                    IF iCurrentCopyY > _RecipeBuilder.ActualCopiesY THEN
                        //Trace(Message := 'Step 90: ZAKONCZONO WSZYSTKIE KOPIE (Nesting gotowy). Skok do 1000.');
                        nStep := 1000;
                    ELSE
                        //Trace(Message := CONCAT('Step 90: Skok do nastepnego rzedu (Kopia Y): ', TO_STRING(iCurrentCopyY)));
                        iCurrentSegment := 1;
                        nStep := 10;
                    END_IF
                ELSE
                    //Trace(Message := CONCAT('Step 90: Skok do nastepnego detalu w rzedzie (Kopia X): ', TO_STRING(iCurrentCopyX)));
                    iCurrentSegment := 1;
                    nStep := 10;
                END_IF
            ELSE
                nStep := 10;
            END_IF
        END_IF

    999: // Błąd
        //Trace(Message := 'Step 999: FATAL ERROR - Aborting');
        _bBusy := FALSE; _bError := TRUE; _bDone := FALSE; nStep := 0;

    1000: // Koniec
        //Trace(Message := 'Step 1000: ZAKONCZONO CALA OPERACJE CIECIA.');
        _bBusy := FALSE; _bDone := TRUE; nStep := 0;
END_CASE
END_METHOD

END_FUNCTION_BLOCK

// ---- POUs/Executor/FB_ExecutorBase.TcPOU
FUNCTION_BLOCK FB_ExecutorBase EXTENDS FB_CyclicFB IMPLEMENTS I_MachiningExecutor, I_BB8Specification
VAR
    // Zmienne sekwencyjne 
    nStep           : INT;
    iCurrentSegment : INT;
    StepTimer       : TON;
    _bBusy          : BOOL;
    _bDone          : BOOL;
    _bError         : BOOL;
    _uErrorID       : UDINT;

    // --- ZMIENNE WSPÓLNE DLA WSZYSTKICH EXECUTORÓW
    _AxisX          : SPT_Motion_Control.I_BasicAxis;
    _AxisY          : SPT_Motion_Control.I_BasicAxis;
    _AxisZ          : SPT_Motion_Control.I_BasicAxis;
	_AxisQ			: SPT_Motion_Control.I_BasicAxis;
    _Cylinder       : I_Cylinder;                     
    _RecipeBuilder  : I_RecipeBuilder;
	_ConfigProvider : I_GantryConfigProvider;
	
	iCurrentCopyX : INT := 1;
    iCurrentCopyY : INT := 1;
END_VAR

METHOD Abort
_bBusy := FALSE;
_bDone := FALSE;
nStep := 0;
iCurrentSegment := 1;
StepTimer(IN := FALSE);
END_METHOD

PROPERTY AxisQ : I_BasicAxis
GET
AxisQ := _AxisQ;
END_GET
SET
_AxisQ := AxisQ;
END_SET
END_PROPERTY

PROPERTY AxisX : I_BasicAxis
GET
AxisX := _AxisX;
END_GET
SET
_AxisX := AxisX;
END_SET
END_PROPERTY

PROPERTY AxisY : I_BasicAxis
GET
AxisY := _AxisY;
END_GET
SET
_AxisY := AxisY;
END_SET
END_PROPERTY

PROPERTY AxisZ : I_BasicAxis
GET
AxisZ := _AxisZ;
END_GET
SET
_AxisZ := AxisZ;
END_SET
END_PROPERTY

PROPERTY Busy : BOOL
GET
Busy := _bBusy;
END_GET
END_PROPERTY

PROPERTY ConfigProvider : I_GantryConfigProvider
GET
ConfigProvider := _ConfigProvider;
END_GET
SET
_ConfigProvider := ConfigProvider;
END_SET
END_PROPERTY

METHOD PUBLIC  CyclicLogic
VAR_INPUT
END_VAR
END_METHOD

PROPERTY Cylinder : I_Cylinder
GET
Cylinder := _Cylinder;
END_GET
SET
_Cylinder := Cylinder;
END_SET
END_PROPERTY

PROPERTY Done : BOOL
GET
Done := _bDone;
END_GET
END_PROPERTY

PROPERTY Error : BOOL
GET
Error := _bError;
END_GET
END_PROPERTY


PROPERTY ErrorID : UDINT
GET
ErrorID := _uErrorID;
END_GET
END_PROPERTY

METHOD Execute : BOOL
IF _bBusy THEN RETURN; END_IF

_bBusy    := TRUE;
_bDone    := FALSE;
_bError   := FALSE;
_uErrorID := 0;
nStep     := 5; 
iCurrentCopyX := 1; 
iCurrentCopyY := 1; 
Execute   := TRUE;
END_METHOD

METHOD PROTECTED MoveToXY 
VAR_INPUT
    TargetX     : REAL; 
    TargetY     : REAL; 
    ToolOffsetX : REAL := 0.0; 
    ToolOffsetY : REAL := 0.0; 
END_VAR
VAR
    localConfig : ST_GantryXYZ_Config;
	NestingOffsetX : REAL;
    NestingOffsetY : REAL;
END_VAR
// Pobieramy bezpieczną konfigurację z Providera (zawiera GlobalOffset)
localConfig := _ConfigProvider.Config;

// Odejmujemy 1, bo pierwsza kopia (indeks 1) ma offset 0.0
NestingOffsetX := (iCurrentCopyX - 1) * _RecipeBuilder.FootprintX;
NestingOffsetY := (iCurrentCopyY - 1) * _RecipeBuilder.FootprintY;

// I dodajemy to do naszych wspaniałych komend jazdy:
_AxisX.MoveAbsolute(TargetX + ToolOffsetX + NestingOffsetX + localConfig.GlobalOffsetX, 0);
_AxisY.MoveAbsolute(TargetY + ToolOffsetY + NestingOffsetY + localConfig.GlobalOffsetY, 0);
END_METHOD

PROPERTY RecipeBuilder : I_RecipeBuilder
GET
RecipeBuilder := _RecipeBuilder;
END_GET
SET
_RecipeBuilder := RecipeBuilder;
END_SET
END_PROPERTY

END_FUNCTION_BLOCK

// ---- POUs/Executor/FB_Exec_Spindle_PTP.TcPOU
FUNCTION_BLOCK FB_Exec_Spindle_PTP EXTENDS FB_ExecutorBase

METHOD PUBLIC CyclicLogic
VAR_INST
    // Lokalne zmienne pomocnicze na czas trwania cyklu
    currentSeg          : ST_CutSegment;
    localConfig         : ST_GantryXYZ_Config;
    recipeConfig        : ST_RecipeBuilder_Config; 
    
    MaterialTopZ        : REAL;
    SafeZ               : REAL;
    TargetZ             : REAL;

    // Zmienne sekwencyjne dla logiki frezowania
    iPass               : INT;
    currentDepth        : LREAL;
    g1, g2, g3, g4, g5  : LREAL;
    v1, v2, v3, v4, v5  : LREAL;
END_VAR
StepTimer();

// Zabezpieczenie na wypadek braku wstrzykniętych referencji!
IF _RecipeBuilder = 0 OR _ConfigProvider = 0 THEN
    RETURN;
END_IF

// Pobieramy konfigurację do pamięci podręcznej 
localConfig := _ConfigProvider.Config;

IF iCurrentSegment < 1 THEN iCurrentSegment := 1; END_IF
IF iCurrentSegment > 32 THEN iCurrentSegment := 32; END_IF

// Wyciągnięcie konkretnego segmentu dla aktualnego kroku
currentSeg := _RecipeBuilder.SegmentsGroove[iCurrentSegment];

// 1. Z=0 to stół. 
// Dodajemy podkład (GlobalOffsetZ) i grubość deski (RawBoardZ).
// To daje nam absolutną pozycję górnej krawędzi płyty w układzie maszyny.
MaterialTopZ := localConfig.GlobalOffsetZ + localConfig.RawBoardZ;

// 2. Pozycja bezpieczna to wierzch płyty + prześwit (np. 10 mm).
// Na tej wysokości możemy latać na parametrze RapidSpeedZ.
SafeZ := MaterialTopZ + localConfig.SafeClearanceZ;

CASE nStep OF
    
    0: // IDLE - maszyna czeka na wywołanie Execute()

    // -------- Inicjalizacja procesu --------
    5:
        // Konfiguracja głębokości (g) i mnożników prędkości (v)
        g1 := 3.5; g2 := 3.5; g3 := 1.5; g4 := 0.0; g5 := 0.0;
        v1 := 1.0; v2 := 1.0; v3 := 1.0; v4 := 1.0; v5 := 1.0;

        IF _AxisX.Enable() AND _AxisY.Enable() AND _AxisZ.Enable() THEN
            IF _RecipeBuilder.SegmentsToGroove <= 0 THEN
                nStep := 1000;
                RETURN;
            END_IF;
           
            _AxisX.Velocity := localConfig.RapidSpeedX;
            _AxisY.Velocity := localConfig.RapidSpeedY;
            _AxisZ.Velocity := localConfig.RapidSpeedZ;

            iCurrentSegment := 1;
            iPass := 4; // Zgodnie z oryginalnym plikiem testowym
            
            IF NOT _AxisX.Busy AND NOT _AxisY.Busy AND NOT _AxisZ.Busy THEN
                nStep := 10;
            END_IF     
        END_IF

    // -------- Dojazd XY do poczatku (Start) --------
    10:
        MoveToXY(currentSeg.Start.X, currentSeg.Start.Y, 0.0, 0.0);
        nStep := 20;

    20: // Czekamy na pozycje XY
        IF _AxisX.Error OR _AxisY.Error THEN 
            nStep := 999;
        ELSIF _AxisX.InPosition AND _AxisY.InPosition THEN 
            _AxisZ.Velocity := localConfig.GroovingSpeedZ;
            nStep := 30;
        END_IF

    // -------- Wybor glebokosci dla przejsc --------
    30:
        recipeConfig := _RecipeBuilder.Config;
        
        CASE iPass OF
            1: currentDepth := recipeConfig.GrooveDepthZ - g1;
            2: currentDepth := recipeConfig.GrooveDepthZ - g2;
            3: currentDepth := recipeConfig.GrooveDepthZ - g3;
            4: currentDepth := recipeConfig.GrooveDepthZ - g4;
            5: currentDepth := recipeConfig.GrooveDepthZ - g5;
        ELSE
            currentDepth := recipeConfig.GrooveDepthZ;
        END_CASE;

        // 3. OBLICZENIE ABSOLUTNEGO CELU DLA OSI Z
        // Skoro MaterialTopZ to góra płyty, a currentDepth to to głębokość,
        // na jaką musimy się w nią zanurzyć - TargetZ = MaterialTopZ - currentDepth.
        TargetZ := MaterialTopZ - currentDepth;
        _AxisZ.MoveAbsolute(TargetZ, 0);
        nStep := 40;

    40: // Czekamy az os Z zjedzie
        IF _AxisZ.Error THEN 
            nStep := 999;
        ELSIF _AxisZ.InPosition THEN
            // Wybor predkosci posuwu roboczego w zaleznosci od przejscia
			// Wybor predkosci posuwu roboczego w zaleznosci od przejscia
            CASE iPass OF
                1: _AxisX.Velocity := localConfig.GroovingSpeedXY * v1; _AxisY.Velocity := localConfig.GroovingSpeedXY * v1;
                2: _AxisX.Velocity := localConfig.GroovingSpeedXY * v2; _AxisY.Velocity := localConfig.GroovingSpeedXY * v2;
                3: _AxisX.Velocity := localConfig.GroovingSpeedXY * v3; _AxisY.Velocity := localConfig.GroovingSpeedXY * v3;
                4: _AxisX.Velocity := localConfig.GroovingSpeedXY * v4; _AxisY.Velocity := localConfig.GroovingSpeedXY * v4;
                5: _AxisX.Velocity := localConfig.GroovingSpeedXY * v5; _AxisY.Velocity := localConfig.GroovingSpeedXY * v5;
            END_CASE;
            
            nStep := 50;
        END_IF
            
    50: // Czekanie przed ruchem
        StepTimer(IN := TRUE, PT := REAL_TO_TIME(localConfig.GroovingIdleTime * 1000.0));
        IF StepTimer.Q THEN
            StepTimer(IN := FALSE);
            nStep := 60;
        END_IF

    // -------- Frezowanie do punktu koncowego --------
    60:
        MoveToXY(currentSeg.Stop.X, currentSeg.Stop.Y, 0.0, 0.0);
        nStep := 70;

    70: // Czekamy na koniec cięcia
        IF _AxisX.Error OR _AxisY.Error OR _AxisZ.Error THEN 
            nStep := 999;
        ELSIF _AxisX.InPosition AND _AxisY.InPosition AND _AxisZ.InPosition THEN
            IF iPass = 5 THEN
                nStep := 74;
            ELSE
                _AxisZ.Velocity := localConfig.RapidSpeedZ;
                nStep := 80;
            END_IF
        END_IF

    // -------- Procedura czyszcząca na koniec 5-go przejazdu --------
    74:
        StepTimer(IN := TRUE, PT := T#500MS);
        IF StepTimer.Q THEN
            StepTimer(IN := FALSE);
            nStep := 75;
        END_IF

    75: 
        MoveToXY(currentSeg.Start.X, currentSeg.Start.Y, 0.0, 0.0);
        nStep := 76;

    76: 
        IF _AxisX.Error OR _AxisY.Error THEN 
            nStep := 999;
        ELSIF _AxisX.InPosition AND _AxisY.InPosition THEN
            _AxisZ.Velocity := localConfig.RapidSpeedZ;
            nStep := 80;
        END_IF

    // -------- Podnoszenie osi Z na pozycję bezpieczną --------
    80:
        // 4. UŻYCIE POZYCJI BEZPIECZNEJ SafeZ 
        // Wcześniej było to sztywne `0`, co stanowiło ryzyko kolizji z materiałem.
        _AxisZ.MoveAbsolute(SafeZ, 0);
        nStep := 90;

    90: 
        IF _AxisZ.Error THEN 
            nStep := 999;
        ELSIF _AxisZ.InPosition THEN
            nStep := 100;
        END_IF  

    100: // Czas stabilizacji po przejsciu
        StepTimer(IN := TRUE, PT := REAL_TO_TIME(localConfig.GroovingIdleTime * 1000.0));
        IF StepTimer.Q THEN
            StepTimer(IN := FALSE);
            
            // Powrot predkosci X/Y na rapid
            _AxisX.Velocity := localConfig.RapidSpeedX;
            _AxisY.Velocity := localConfig.RapidSpeedY;
            iCurrentSegment := iCurrentSegment + 1;
            
            // Logika zmiany przejazdu / zakonczenia
            IF iCurrentSegment > _RecipeBuilder.SegmentsToGroove THEN
                IF iPass < 5 THEN
                    iPass := iPass + 1;
                    iCurrentSegment := 1;
                    nStep := 10;
                ELSE
                    // CZYSTA PĘTLA NESTINGU (Zrobiono wszystkie 5 passów)
                    iCurrentCopyX := iCurrentCopyX + 1;
                    
                    IF iCurrentCopyX > _RecipeBuilder.ActualCopiesX THEN
                        iCurrentCopyX := 1;
                        iCurrentCopyY := iCurrentCopyY + 1;
                        
                        IF iCurrentCopyY > _RecipeBuilder.ActualCopiesY THEN
                            nStep := 1000;
                        ELSE
                            iPass := 1;
                            iCurrentSegment := 1;
                            nStep := 10;
                        END_IF
                    ELSE
                        iPass := 1;
                        iCurrentSegment := 1;
                        nStep := 10;
                    END_IF
                END_IF
            ELSE
                nStep := 10;
            END_IF
        END_IF

    999: // Błąd którejkolwiek osi
        _bBusy  := FALSE;
        _bError := TRUE; 
        _bDone  := FALSE;
        nStep   := 0;

    1000: // Zakonczenie operacji frezowania
        _bBusy := FALSE;
        _bDone := TRUE;
        nStep := 0;
END_CASE
END_METHOD

END_FUNCTION_BLOCK

// ---- POUs/Executor/FB_Exec_Drill_PTP.TcPOU
FUNCTION_BLOCK FB_Exec_Drill_PTP EXTENDS FB_ExecutorBase

METHOD PUBLIC CyclicLogic
VAR_INST
    currentHole   : ST_PointXY;
    localConfig   : ST_GantryXYZ_Config;
    recipeConfig  : ST_RecipeBuilder_Config;
    
    MaterialTopZ  : REAL;
    SafeZ         : REAL;
    TargetZ       : REAL;
END_VAR
// 1. Zabezpieczenia i cykliczny timer z klasy bazowej
StepTimer();
IF _RecipeBuilder = 0 OR _ConfigProvider = 0 OR _AxisQ = 0 THEN RETURN; END_IF

// 2. Cache'owanie danych wejściowych
localConfig := _ConfigProvider.Config;

// Zabezpieczenie zakresu tablicy
IF iCurrentSegment < 1 THEN iCurrentSegment := 1; END_IF
IF iCurrentSegment > 1000 THEN iCurrentSegment := 1000; END_IF

currentHole := _RecipeBuilder.HolesDrill[iCurrentSegment];

// 3. Oliczenie bezpiecznych poziomów w osi Z 
MaterialTopZ := localConfig.GlobalOffsetZ + localConfig.RawBoardZ;
SafeZ := MaterialTopZ + localConfig.SafeClearanceZ;

CASE nStep OF
    0: // IDLE

    5: // INIT - Aktywacja osi i przygotowanie (X, Y, Z oraz Q!)
        IF _AxisX.Enable() AND _AxisY.Enable() AND _AxisZ.Enable() AND _AxisQ.Enable() THEN
            IF _RecipeBuilder.HolesToDrill <= 0 THEN
                nStep := 1000; // Brak otworów do wiercenia
                RETURN;
            END_IF;
           
            _AxisX.Velocity := localConfig.RapidSpeedX;
            _AxisY.Velocity := localConfig.RapidSpeedY;
            _AxisZ.Velocity := localConfig.RapidSpeedZ;
            _AxisQ.Velocity := localConfig.RapidSpeedQ; // Ustawienie prędkosci noża

            iCurrentSegment := 1;
            nStep := 6;
      END_IF
	  
	6:
		IF NOT _AxisX.Busy AND NOT _AxisY.Busy AND NOT _AxisZ.Busy AND NOT _AxisQ.Busy THEN
			nStep := 10;
		END_IF   

    // -------- Dojazd XY nad punkt otworu --------
    10:
        MoveToXY(currentHole.X, currentHole.Y, 0.0, 0.0);
        nStep := 20;

    20: // Czekamy na pozycje XY
        IF _AxisX.Error OR _AxisY.Error THEN 
            nStep := 999;
        ELSIF _AxisX.InPosition AND _AxisY.InPosition THEN 
            // Ustawiamy prędkość roboczą dla zagłębiania noża
            _AxisZ.Velocity := localConfig.GroovingSpeedZ;
            nStep := 30;
        END_IF

    // -------- Zjazd Z (Zanurzenie noża w gąbce) --------
    30:
        recipeConfig := _RecipeBuilder.Config;
        TargetZ := MaterialTopZ - 2.0;
        _AxisZ.MoveAbsolute(TargetZ, 0);
        nStep := 40;

    40: // Czekamy aż nóż wejdzie w materiał
        IF _AxisZ.Error THEN 
            nStep := 999;
        ELSIF _AxisZ.InPosition THEN
            // Zjechaliśmy! Teraz kręcimy nożem tangencjalnym do 720 stopni
            _AxisQ.MoveAbsolute(720.0, 0);
            nStep := 42;
        END_IF
        
    // -------- Obrót Q: Piruet otworowy --------
    42: // Czekamy aż nóż osiągnie +720 stopni
        IF _AxisQ.Error THEN
            nStep := 999;
        ELSIF _AxisQ.InPosition THEN
            // Wracamy nożem do 0 stopni, żeby nie zrywać przewodów/pasków
            _AxisQ.MoveAbsolute(0.0, 0);
            nStep := 44;
        END_IF
        
    44: // Czekamy aż nóż wróci do 0
        IF _AxisQ.Error THEN
            nStep := 999;
        ELSIF _AxisQ.InPosition THEN
            nStep := 50;
        END_IF
            
    50: // Czekanie na dnie otworu (Opcjonalne uspokojenie materiału po obrocie)
        StepTimer(IN := TRUE, PT := REAL_TO_TIME(localConfig.GroovingIdleTime * 1000.0));
        IF StepTimer.Q THEN
            StepTimer(IN := FALSE);
            nStep := 60;
        END_IF

    // -------- Szybki wyjazd z materiału --------
    60:
        _AxisZ.Velocity := localConfig.RapidSpeedZ;
        _AxisZ.MoveAbsolute(SafeZ, 0);
        nStep := 70;

    70: // Czekamy na wyjazd osi Z
        IF _AxisZ.Error THEN 
            nStep := 999;
        ELSIF _AxisZ.InPosition THEN
            // Krok zakończony - idziemy do następnego otworu
            iCurrentSegment := iCurrentSegment + 1;
            
            IF iCurrentSegment > _RecipeBuilder.HolesToDrill THEN
                // CZYSTA PĘTLA NESTINGU
                iCurrentCopyX := iCurrentCopyX + 1;
                
                IF iCurrentCopyX > _RecipeBuilder.ActualCopiesX THEN
                    iCurrentCopyX := 1;
                    iCurrentCopyY := iCurrentCopyY + 1;
                    
                    IF iCurrentCopyY > _RecipeBuilder.ActualCopiesY THEN
                        // Wiercenie wszystkich kopii zakończone
                        nStep := 1000;
                    ELSE
                        iCurrentSegment := 1;
                        nStep := 10;
                    END_IF
                ELSE
                    iCurrentSegment := 1;
                    nStep := 10;
                END_IF
            ELSE
                nStep := 10;
            END_IF
        END_IF

    // -------- Awaria --------
    999: 
        _bBusy  := FALSE;
        _bError := TRUE; 
        _bDone  := FALSE;
        nStep   := 0;
        
    // -------- Sukces --------
    1000: 
        _bBusy := FALSE;
        _bDone := TRUE;
        nStep := 0;
END_CASE
END_METHOD

END_FUNCTION_BLOCK

// ---- POUs/Executor/FB_Exec_Tangential_FeedTable.TcPOU
FUNCTION_BLOCK FB_Exec_Tangential_FeedTable EXTENDS FB_ExecutorBase IMPLEMENTS I_GeometryWriter
VAR
    _NciChannel : I_NciChannel_FeedTable;
    _FeedTable  : ST_NciFeedGroupTable; 
    
    // NCI Builder z Tc2_PlcInterpolation
    fbFeedPrep  : FB_NciFeedTablePreparation;
	
	// Lokalne offsety aktualizowane co kopię nestingu
	_CurrentOffsetX : LREAL;
	_CurrentOffsetY : LREAL;
END_VAR

METHOD Abort
IF _NciChannel <> 0 THEN
    _NciChannel.Stop();
    _NciChannel.ResetChannel();
    _NciChannel.Ungroup();
END_IF
_bBusy := FALSE; _bDone := FALSE; _bError := FALSE; _uErrorID := 0; nStep := 0;
END_METHOD

METHOD AddArc : BOOL
VAR_INPUT
    TargetX    : LREAL;
    TargetY    : LREAL;
    CenterX    : LREAL;
    CenterY    : LREAL;
    Velo       : LREAL;
    Clockwise  : BOOL; 
END_VAR
VAR
    stArc : ST_NciGeoCirclePlane;
END_VAR
stArc.fEndPosX := TargetX + _CurrentOffsetX;
stArc.fEndPosY := TargetY + _CurrentOffsetY;
stArc.fCenterX := CenterX + _CurrentOffsetX;
stArc.fCenterY := CenterY + _CurrentOffsetY;
stArc.fVelo := Velo;
stArc.bClockwise := Clockwise;
stArc.nPlane := E_NciGeoPlane.E_NciGeoPlaneXY;

fbFeedPrep(
    nEntryType := E_NciEntryType.E_NciEntryTypeGeoCirclePlane,
    pEntry := ADR(stArc),
    bResetTable := FALSE,
    bResetAll := FALSE,
    stFeedGroupTable := _FeedTable
);
AddArc := NOT fbFeedPrep.bError;
END_METHOD

METHOD AddLine : BOOL
VAR_INPUT
    TargetX : LREAL;
    TargetY : LREAL;
    Velo    : LREAL;
END_VAR
VAR
    stLine : ST_NciGeoLine;
END_VAR
stLine.fEndPosX := TargetX + _CurrentOffsetX;
stLine.fEndPosY := TargetY + _CurrentOffsetY;
stLine.fVelo := Velo;

fbFeedPrep(
    nEntryType := E_NciEntryType.E_NciEntryTypeGeoLine,
    pEntry := ADR(stLine),
    bResetTable := FALSE,
    bResetAll := FALSE,
    stFeedGroupTable := _FeedTable
);
AddLine := NOT fbFeedPrep.bError;
END_METHOD

METHOD AddStartPoint : BOOL
VAR_INPUT
    TargetX : LREAL;
    TargetY : LREAL;
END_VAR
VAR
    stStart : ST_NciGeoStart;
END_VAR
stStart.fPosX := TargetX + _CurrentOffsetX;
stStart.fPosY := TargetY + _CurrentOffsetY;

fbFeedPrep(
    nEntryType := E_NciEntryType.E_NciEntryTypeGeoStart,
    pEntry := ADR(stStart),
    bResetTable := FALSE,
    bResetAll := FALSE,
    stFeedGroupTable := _FeedTable
);
AddStartPoint := NOT fbFeedPrep.bError;
END_METHOD

METHOD Clear : BOOL
VAR_INPUT
END_VAR
fbFeedPrep(
    nEntryType := E_NciEntryType.E_NciEntryTypeNone,
    pEntry := 0,
    bResetTable := TRUE,
    bResetAll := TRUE, // Czyści też modale i błędy (wg str. 315)
    stFeedGroupTable := _FeedTable
);
Clear := NOT fbFeedPrep.bError;
END_METHOD

METHOD PUBLIC CyclicLogic
VAR_INST
    localConfig   : ST_GantryXYZ_Config;
    recipeConfig  : ST_RecipeBuilder_Config;
    MaterialTopZ  : REAL;
    SafeZ         : REAL;
    TargetZ       : REAL;
    iCurrentShape : INT := 1;
END_VAR
SUPER^.CyclicLogic();

IF nStep > 0 THEN
    IF _RecipeBuilder = 0 OR _ConfigProvider = 0 OR _NciChannel = 0 THEN
        nStep := 999;
    END_IF
END_IF

CASE nStep OF
    0: 
		;
    5: 
        IF _AxisX.Enable() AND _AxisY.Enable() AND _AxisZ.Enable() AND _AxisQ.Enable() THEN
            IF _AxisX.Enabled AND _AxisY.Enabled AND _AxisZ.Enabled AND _AxisQ.Enabled 
               AND NOT _AxisX.Busy AND NOT _AxisY.Busy AND NOT _AxisQ.Busy THEN
                
                _bBusy := TRUE;
                localConfig := _ConfigProvider.Config;
                recipeConfig := _RecipeBuilder.Config;

                IF NOT recipeConfig.IsValid THEN
                    nStep := 1000;
                    RETURN;
                END_IF

                iCurrentCopyX := 1;
                iCurrentCopyY := 1;
                iCurrentShape := 1;

                _AxisX.Velocity := localConfig.RapidSpeedX;
                _AxisY.Velocity := localConfig.RapidSpeedY;
                _AxisZ.Velocity := localConfig.RapidSpeedZ;
                _AxisQ.Velocity := localConfig.RapidSpeedQ;

                nStep := 8;
            END_IF
        END_IF

    8: 
        localConfig := _ConfigProvider.Config;
		_CurrentOffsetX := (iCurrentCopyX - 1) * _RecipeBuilder.FootprintX + localConfig.GlobalOffsetX;
		_CurrentOffsetY := (iCurrentCopyY - 1) * _RecipeBuilder.FootprintY + localConfig.GlobalOffsetY;
		
        _RecipeBuilder.CurrentShapeIndex := iCurrentShape;
		_RecipeBuilder.Build();
		nStep := 85;

	85:
		IF _RecipeBuilder.Done THEN
			recipeConfig := _RecipeBuilder.Config;
			MoveToXY(_RecipeBuilder.ShapeStart[iCurrentShape].X, _RecipeBuilder.ShapeStart[iCurrentShape].Y, 0.0, 0.0);
			_AxisQ.MoveAbsolute(0.0, 0);
			nStep := 9;
		ELSIF _RecipeBuilder.Error THEN
			nStep := 999;
		END_IF

    9: 
        IF _AxisX.Error OR _AxisY.Error OR _AxisZ.Error OR _AxisQ.Error THEN
            nStep := 999;
        ELSIF _AxisX.InPosition AND _AxisY.InPosition AND NOT _AxisQ.Busy THEN
            localConfig := _ConfigProvider.Config;
            MaterialTopZ := localConfig.GlobalOffsetZ + localConfig.RawBoardZ;
            SafeZ := MaterialTopZ + localConfig.SafeClearanceZ;

            IF _AxisZ.MoveAbsolute(SafeZ, 0) THEN
                nStep := 10;
            END_IF
        END_IF

    10: 
        IF _AxisZ.Error THEN
            nStep := 999;
        ELSIF _AxisZ.InPosition THEN
            nStep := 20;
        END_IF

    20: 
        _NciChannel.BuildGroup();
        nStep := 30;

    30: 
        IF _NciChannel.ChannelError THEN
            nStep := 999;
        ELSIF _NciChannel.IsGrouped THEN
            TargetZ := MaterialTopZ - recipeConfig.GrooveDepthZ;
            _AxisZ.Velocity := localConfig.GroovingSpeedZ;
			IF  _AxisZ.MoveAbsolute(TargetZ, 0) THEN
				nStep := 35;
			END_IF
        END_IF

    35: 
        IF _AxisZ.Error THEN
            nStep := 999;
        ELSIF _AxisZ.InPosition THEN
            _NciChannel.StartFeedTable(stTable := THIS^._FeedTable); 
            nStep := 40;
        END_IF

    40: 
        IF _NciChannel.ChannelError THEN
            nStep := 999;
        ELSIF _NciChannel.IsFeedingDone THEN
            nStep := 50;
        END_IF

    50: 
        IF _NciChannel.ChannelError THEN
            nStep := 999;
        ELSIF _NciChannel.IsChannelDone THEN
            _AxisZ.Velocity := localConfig.RapidSpeedZ;
            _AxisZ.MoveAbsolute(SafeZ, 0);
            nStep := 55;
        END_IF

    55:
        IF _AxisZ.Error THEN
            nStep := 999;
        ELSIF _AxisZ.InPosition THEN
            _NciChannel.ResetChannel();
            nStep := 80;
        END_IF

    80: 
        _NciChannel.Ungroup();
        nStep := 90;

    90: 
        IF NOT _NciChannel.IsGrouped THEN
            iCurrentShape := iCurrentShape + 1;
            IF iCurrentShape > _RecipeBuilder.ShapesCount THEN
                iCurrentShape := 1;
                nStep := 110;
            ELSE
                nStep := 8;
            END_IF
        END_IF

    110:
        iCurrentCopyX := iCurrentCopyX + 1;
        IF iCurrentCopyX > _RecipeBuilder.ActualCopiesX THEN
            iCurrentCopyX := 1;
            iCurrentCopyY := iCurrentCopyY + 1;
            IF iCurrentCopyY > _RecipeBuilder.ActualCopiesY THEN
                nStep := 1000;
            ELSE
                nStep := 8;
            END_IF
        ELSE
            nStep := 8;
        END_IF

    999: 
        _bBusy := FALSE;
        _bError := TRUE;
        _bDone := FALSE;
        _uErrorID := _NciChannel.ChannelErrorId;
        _NciChannel.Ungroup();
        nStep := 0;

    1000: 
        _bBusy := FALSE;
        _bDone := TRUE;
        nStep := 0;
END_CASE
END_METHOD

METHOD EnableTangentialFollowing : BOOL
VAR
    stTf : ST_NciTangentialFollowingDesc;
END_VAR
stTf.bTangOn := TRUE;
stTf.nTangAxis := E_NciAxesInGroup.Q1Axis;
stTf.nPathAxis1 := E_NciAxesInGroup.XAxis;
stTf.nPathAxis2 := E_NciAxesInGroup.YAxis;
stTf.fOffset := -90.0;
stTf.fCriticalAngle1 := 90.0; 
stTf.nTfBehavior := E_TangentialFollowingBehavior.E_TfIngoreAll; // Uwaga na literówkę Beckhoffa!

fbFeedPrep(
    nEntryType := E_NciEntryType.E_NciEntryTypeTfDesc,
    pEntry := ADR(stTf),
    bResetTable := FALSE,
    bResetAll := FALSE,
    stFeedGroupTable := _FeedTable
);
EnableTangentialFollowing := NOT fbFeedPrep.bError;
END_METHOD

METHOD EndTable : BOOL
VAR
    stEnd : ST_NciEndOfTables;
END_VAR

fbFeedPrep(
    nEntryType := E_NciEntryType.E_NciEntryTypeEndOfTables,
    pEntry := ADR(stEnd),
    bResetTable := FALSE,
    bResetAll := FALSE,
    stFeedGroupTable := _FeedTable
);
EndTable := NOT fbFeedPrep.bError;
END_METHOD

PROPERTY NciChannel : I_NciChannel_FeedTable
GET
NciChannel := _NciChannel;
END_GET
SET
_NciChannel := NciChannel;
END_SET
END_PROPERTY

END_FUNCTION_BLOCK

// ---- POUs/Executor/FB_Exec_Spindle_GCodeXYZ.TcPOU
FUNCTION_BLOCK FB_Exec_Spindle_GCodeXYZ EXTENDS FB_ExecutorBase
VAR
    _NciChannel : I_NciChannel_GCode;
END_VAR

METHOD Abort
// 1. Zatrzymujemy program NCI (jeśli jedzie)
_NciChannel.Stop();

// 2. Wymuszamy reset błędów na kanale interpolacyjnym
_NciChannel.ResetChannel();

// 3. Dopiero teraz bezpiecznie nakazujemy kanałowi rozpięcie grupy
_NciChannel.Ungroup();

// 4. Zerujemy resztę lokalnych zmiennych Executora
_bBusy := FALSE;
_bDone := FALSE;
_bError := FALSE;
_uErrorID := 0;
nStep := 0;
iCurrentSegment := 1;
StepTimer(IN := FALSE);
END_METHOD

METHOD PUBLIC CyclicLogic
VAR_INST

    refX : Tc2_MC2.AXIS_REF;
    refY : Tc2_MC2.AXIS_REF;
    refZ : Tc2_MC2.AXIS_REF;
    
	MaterialTopZ : REAL;
    SafeZ        : REAL;

    recipeConfig  : ST_RecipeBuilder_Config;
    machineConfig : ST_GantryXYZ_Config;
END_VAR
// --- LOGIKA ---
StepTimer();

// Zabezpieczenie przed brakiem wstrzykniętych referencji
IF nStep > 0 THEN
	IF _RecipeBuilder = 0 OR _ConfigProvider = 0 OR _NciChannel = 0 OR _AxisX = 0 OR _AxisY = 0 OR _AxisZ = 0 OR _AxisQ = 0 THEN
		IF nStep > 0 THEN
			ADSLOGSTR(ADSLOG_MSGTYPE_ERROR, 'ExecutorNCI: BRAK KRYTYCZNYCH REFERENCJI (Builder/Provider/NCI/Osie)!', '');
			nStep := 999;
		END_IF
		RETURN; 
	END_IF
END_IF

CASE nStep OF
    0: // IDLE

	5: // INIT - Załączanie osi i start
		IF _AxisX.Enable() AND _AxisY.Enable() AND _AxisZ.Enable() AND _AxisQ.Enable() THEN 
			IF _AxisX.Error OR _AxisY.Error OR _AxisZ.Error OR _AxisQ.Error THEN 
				nStep := 999;
			ELSIF _AxisX.Enabled AND _AxisY.Enabled AND _AxisZ.Enabled AND _AxisQ.Enabled THEN 
				_bBusy := TRUE;
								 
				// Odczyt właściwości (Properties) do lokalnych zmiennych pomocniczych!
				machineConfig := _ConfigProvider.Config;
				recipeConfig  := _RecipeBuilder.Config;
								 
				// Bezpieczne użycie zmiennych lokalnych
				_AxisX.Velocity := machineConfig.RapidSpeedX;
				_AxisY.Velocity := machineConfig.RapidSpeedY;
				_AxisZ.Velocity := machineConfig.RapidSpeedZ;
				_AxisQ.Velocity := machineConfig.RapidSpeedQ; // <-- DODANO Q
											 
				nStep := 8;
			END_IF
		END_IF

	8: // 1. Dojazd PTP do punktu startowego NCI
       
        nStep := 9;

	9: 
		IF _AxisX.Error OR _AxisY.Error OR _AxisZ.Error OR _AxisQ.Error THEN 
			nStep := 999;
		ELSIF _AxisX.InPosition AND _AxisY.InPosition THEN
			
			machineConfig := _ConfigProvider.Config;
			
			_AxisQ.MoveAbsolute(0,0);

			nStep := 10;
		END_IF
        
    10: // Czekamy aż podniesie się Z
        IF _AxisQ.Error THEN
            nStep := 999;
        ELSIF _AxisQ.InPosition THEN
            nStep := 20;
        END_IF

	20: // 2. Zbudowanie grupy NCI
		_NciChannel.BuildGroup();
		nStep := 30;

    30: // Czekamy na spięcie osi
        IF _NciChannel.ChannelError THEN 
            nStep := 999;
        ELSIF _NciChannel.IsGrouped THEN 
            nStep := 40; 
        END_IF

    40: // 3. Załadowanie pliku G-Code
        recipeConfig := _RecipeBuilder.Config;
        _NciChannel.LoadProgram(recipeConfig.GCodePath);
        nStep := 50;

    50: // Czekamy na załadowanie do bufora
        IF _NciChannel.ChannelError THEN 
            nStep := 999;
        ELSIF _NciChannel.IsProgramLoaded THEN 
            nStep := 60;
        END_IF

    60: // 4. START programu CNC!
        _NciChannel.Start();
        StepTimer(IN:=FALSE);
        nStep := 70;
	
	70: // 4. Czekamy na koniec programu (M30)
        IF _NciChannel.ChannelError THEN 
            nStep := 999;
        ELSIF _NciChannel.IsReady THEN 
            ADSLOGSTR(ADSLOG_MSGTYPE_HINT, 'Executor: Program NCI zakonczony (M30). Rozpinam grupe...', '');
            nStep := 80;
        END_IF

    80: // 5. Rozwiązanie grupy, uwalniamy osie z powrotem do trybu PTP
        _NciChannel.Ungroup();
        nStep := 90;

	90: // 6. Reset kanału i zakończenie pracy
        IF NOT _NciChannel.IsGrouped THEN
            ADSLOGSTR(ADSLOG_MSGTYPE_HINT, 'Executor: Osie uwolnione do trybu PTP. Resetuje kanal.', '');
            _NciChannel.ResetChannel(); 
            
            nStep := 1000; 
        END_IF
        
    999: // ERROR HANDLING
        _bBusy := FALSE;
        _bError := TRUE;
        _bDone := FALSE;
        _uErrorID := _NciChannel.ChannelErrorId;
        ADSLOGDINT(ADSLOG_MSGTYPE_ERROR, 'Executor: BLAD KRYTYCZNY NCI! Kod bledu: %d', UDINT_TO_DINT(_uErrorID));
        _NciChannel.Ungroup();
        nStep := 0;

    1000: // ZAKOŃCZONO SUKCESEM
        ADSLOGSTR(ADSLOG_MSGTYPE_HINT, 'ExecutorNCI: Program wykonany pomyslnie.', '');
        _bBusy := FALSE;
        _bDone := TRUE;
        nStep := 0;

END_CASE
END_METHOD

PROPERTY NciChannel : I_NciChannel_GCode
GET
NciChannel := _NciChannel;
END_GET
SET
_NciChannel := NciChannel;
END_SET
END_PROPERTY

END_FUNCTION_BLOCK

// ---- POUs/Components/FB_NciChannel.TcPOU
FUNCTION_BLOCK FB_NciChannel EXTENDS FB_ComponentBase IMPLEMENTS I_NciChannel_GCode

VAR_INPUT
    stAxisIds : ST_NciAxisIds;
	nGroupId  : UDINT := 4;
END_VAR

VAR
    // Zmienne zlinkowane bezpośrednio z hardwarem kanału NCI
    stNciToPlc AT %I* : NCTOPLC_NCICHANNEL_REF; 
    stPlcToNci AT %Q* : PLCTONC_NCICHANNEL_REF;

    // Bloki systemowe Beckhoffa do obsługi grupy
	fbBuildExtGroup : CfgBuildExt3DGroup;
    fbUngroup       : CfgReconfigGroup;
    
    // Bloki systemowe do obsługi programu i ruchu (nowe wersje Ex)
    fbLoadProg      : ItpLoadProgEx;
    fbStartStop     : ItpStartStopEx;
    fbReset         : ItpResetEx2;
    
    _IsGrouped      : BOOL;
    _IsProgLoaded   : BOOL;
    _IsReady		:BOOL;
	


END_VAR

METHOD BuildGroup
_IsGrouped := FALSE;
_Error := FALSE; 
_ErrorId := 0;

fbBuildExtGroup(
    bExecute := TRUE,
    nGroupId := nGroupId,
    nXAxisId := stAxisIds.nX,
    nYAxisId := stAxisIds.nY,
    nZAxisId := stAxisIds.nZ,
    nQ1AxisId := stAxisIds.nQ1
);
END_METHOD

PROPERTY ChannelError : BOOL
GET
ChannelError := _Error OR (stNciToPlc.ErrorCode <> 0);
END_GET
END_PROPERTY

PROPERTY ChannelErrorId : UDINT
GET
IF stNciToPlc.ErrorCode <> 0 THEN
    ChannelErrorId := stNciToPlc.ErrorCode;
ELSE
    ChannelErrorId := _ErrorId;
END_IF
END_GET
END_PROPERTY

// This method serves as the entry point for all underlying FB logic
METHOD PUBLIC CyclicLogic

// This method should be called cyclically by descendant function blocks by invoking SUPER^.CyclicLogic().  Alternatively, the contents of this method could be reimplemented entirely in which case a call to this method would not be necessary.
// Wywołanie bazowe
SUPER^.CyclicLogic();

// Odblokowanie posuwu kanału NCI (1000000 = 100%)
stPlcToNci.ChnAxesOvr := 1000000;

// --- ODŚWIEŻANIE BLOKÓW SYSTEMOWYCH ---
fbBuildExtGroup(tTimeOut := T#2S);
fbUngroup(tTimeOut := T#2S);


fbLoadProg(
    sNciToPlc := stNciToPlc, 
    tTimeOut := T#2S
);

fbStartStop(
    sNciToPlc := stNciToPlc, 
    tTimeOut := T#2S
);

fbReset(
    sNciToPlc := stNciToPlc, 
    tTimeOut := T#2S
);

// --- AKTUALIZACJA STATUSÓW ---
// Obsługa stanów dla tworzenia grupy
IF fbStartStop.bErr THEN
    _Error := TRUE;
    _ErrorId := fbStartStop.nErrId;
    fbStartStop(bStart := FALSE, bStop := FALSE, sNciToPlc := stNciToPlc);
ELSIF fbStartStop.bBusy THEN
    // Skoro kanał NCI przyjął komendę i jest zajęty, opuszczamy Start, 
    // aby przygotować blok na kolejne uruchomienie w przyszłości
    fbStartStop(bStart := FALSE, sNciToPlc := stNciToPlc);
ELSIF NOT fbStartStop.bBusy AND fbStartStop.bStop THEN
    // Jak się poprawnie zatrzymał, opuszczamy flagę Stop
    fbStartStop(bStop := FALSE, sNciToPlc := stNciToPlc);
END_IF

// Obsługa stanów dla rozpinania grupy
IF fbUngroup.bErr THEN
    _Error := TRUE;
    _ErrorId := fbUngroup.nErrId;
    fbUngroup(bExecute := FALSE);
    _IsGrouped := FALSE; // W razie błędu awaryjnie zdejmujemy flagę, żeby maszyna nie utknęła na zawsze
ELSIF fbUngroup.bBusy = FALSE AND fbUngroup.bExecute THEN
    _IsGrouped := FALSE; // Pomyślnie rozpięto!
    fbUngroup(bExecute := FALSE);
END_IF


IF fbBuildExtGroup.bErr THEN
    _Error := TRUE;
    _ErrorId := fbBuildExtGroup.nErrId;
ELSIF fbBuildExtGroup.bBusy = FALSE AND fbBuildExtGroup.bExecute THEN
    _IsGrouped := TRUE;
    fbBuildExtGroup(bExecute := FALSE);
END_IF

// Podobnie dla ładowania programu
IF fbLoadProg.bErr THEN
    _Error := TRUE;
    _ErrorId := fbLoadProg.nErrId;
ELSIF fbLoadProg.bBusy = FALSE AND fbLoadProg.bExecute THEN
    _IsProgLoaded := TRUE;
	fbLoadProg(bExecute := FALSE, sNciToPlc := stNciToPlc);
END_IF

// --- OBSŁUGA ZEROWANIA fbReset ---
IF fbReset.bErr THEN
    _Error := TRUE;
    _ErrorId := fbReset.nErrId;
    fbReset(bExecute := FALSE, sNciToPlc := stNciToPlc);
ELSIF fbReset.bBusy = FALSE AND fbReset.bExecute THEN
    fbReset(bExecute := FALSE, sNciToPlc := stNciToPlc);
END_IF
END_METHOD

PROPERTY IsGrouped : BOOL
GET
IsGrouped := _IsGrouped;
END_GET
END_PROPERTY

PROPERTY IsMoving : BOOL
GET
IsMoving := (stNciToPlc.ItpState = 5);
END_GET
END_PROPERTY

PROPERTY IsProgramLoaded : BOOL
GET
IsProgramLoaded := _IsProgLoaded;
END_GET
END_PROPERTY

PROPERTY IsReady : BOOL
GET
IsReady := (stNciToPlc.ItpState = 2);
END_GET
END_PROPERTY

METHOD LoadProgram
VAR_INPUT
	sProgramPath : STRING(255);
END_VAR
_IsProgLoaded := FALSE;
fbLoadProg(
    bExecute := TRUE,
    sPrg := sProgramPath,
    nLength := INT_TO_UDINT(LEN(sProgramPath)),
    sNciToPlc := stNciToPlc 
);
END_METHOD

METHOD ResetChannel
VAR_INPUT
END_VAR
// Najpierw bezwarunkowo ubijamy flagi ruchu
fbStartStop(bStart := FALSE, bStop := FALSE, sNciToPlc := stNciToPlc);

// Następnie resetujemy sam kanał NCI
fbReset(
    bExecute := TRUE,
    sNciToPlc := stNciToPlc
);

_Error := FALSE;
_ErrorId := 0;
END_METHOD

METHOD Start
VAR_INPUT
END_VAR
fbStartStop(
    bStart := TRUE, 
    bStop := FALSE,
    sNciToPlc := stNciToPlc 
);
END_METHOD

METHOD Stop
VAR_INPUT
END_VAR
fbStartStop(
    bStart := FALSE, 
    bStop := TRUE,
    sNciToPlc := stNciToPlc
);
END_METHOD

METHOD Ungroup
VAR_INPUT
END_VAR
fbUngroup(
    bExecute := TRUE, 
    nGroupId := nGroupId
);
END_METHOD

END_FUNCTION_BLOCK

// ---- POUs/Components/FB_NciChannelTangential.TcPOU
FUNCTION_BLOCK FB_NciChannelTangential EXTENDS FB_ComponentBase IMPLEMENTS I_NciChannel_FeedTable

VAR_INPUT
    stAxisIds : ST_NciAxisIds;
	nGroupId  : UDINT := 5;
END_VAR

VAR
    stNciToPlc AT %I* : NCTOPLC_NCICHANNEL_REF;
    stPlcToNci AT %Q* : PLCTONC_NCICHANNEL_REF;
	
    // ZMIANA: Blok Ext3DGroup pozwala dodać osie Q1..Q5
    fbBuildExtGroup : CfgBuildExt3DGroup;
    fbUngroup       : CfgReconfigGroup;
    
    // Obsługa Resetu / Start / Stop
    fbStartStop     : ItpStartStopEx;
    fbReset         : ItpResetEx2;

    // --- NOWOŚĆ: Blok do przesyłania tabel z RAMu ---
    fbFeedTable     : FB_NciFeedTable;
    refFeedTable    : REFERENCE TO ST_NciFeedGroupTable; // Przechowuje wskaźnik do tabeli z Executora
    _bExecuteFeed   : BOOL;
    _IsFeedingDone  : BOOL;
    _IsChannelDone  : BOOL;

    _IsGrouped      : BOOL;
    _IsReady		: BOOL;
	
	_bResetFeed : BOOL;
END_VAR

METHOD BuildGroup
_IsGrouped := FALSE;
_Error := FALSE; 
_ErrorId := 0;

fbBuildExtGroup(
    bExecute := TRUE,
    nGroupId := nGroupId,
    nXAxisId := stAxisIds.nX,
    nYAxisId := stAxisIds.nY,
    nZAxisId := stAxisIds.nZ,
    nQ1AxisId := stAxisIds.nQ1 
);
END_METHOD

PROPERTY ChannelError : BOOL
GET
ChannelError := _Error OR (stNciToPlc.ErrorCode <> 0);
END_GET
END_PROPERTY

PROPERTY ChannelErrorId : UDINT
GET
IF stNciToPlc.ErrorCode <> 0 THEN
    ChannelErrorId := stNciToPlc.ErrorCode;
ELSE
    ChannelErrorId := _ErrorId;
END_IF
END_GET
END_PROPERTY

METHOD PUBLIC CyclicLogic
SUPER^.CyclicLogic();


stPlcToNci.ChnAxesOvr := 1000000;


fbBuildExtGroup(tTimeOut := T#2S);
fbUngroup(tTimeOut := T#2S);
fbStartStop(sNciToPlc := stNciToPlc, tTimeOut := T#2S);
fbReset(sNciToPlc := stNciToPlc, tTimeOut := T#2S);


IF __ISVALIDREF(refFeedTable) THEN
    fbFeedTable(
        bExecute := _bExecuteFeed,
        bReset := _bResetFeed,
        stFeedGroupTable := refFeedTable,
        stNciToPlc := stNciToPlc,
        bFeedingDone => _IsFeedingDone,
        bChannelDone => _IsChannelDone
    );
    
 
    IF _bResetFeed THEN
        _bResetFeed := FALSE;
    END_IF


    IF _IsChannelDone OR fbFeedTable.bError THEN
        IF _bExecuteFeed AND _IsChannelDone THEN
            ADSLOGSTR(ADSLOG_MSGTYPE_HINT, 'NciChannelTan: Ruch interpolowany zakonczony (Channel Done).', '');
        END_IF
        _bExecuteFeed := FALSE;
    END_IF
    
    IF fbFeedTable.bError THEN
        IF NOT _Error THEN
            ADSLOGDINT(ADSLOG_MSGTYPE_ERROR, 'NciChannelTan: BLAD FeedTable! Kod: %d', UDINT_TO_DINT(fbFeedTable.nErrorId));
        END_IF
        _Error := TRUE;
        _ErrorId := fbFeedTable.nErrorId;
    END_IF
END_IF


IF fbStartStop.bErr THEN
    IF NOT _Error THEN
        ADSLOGDINT(ADSLOG_MSGTYPE_ERROR, 'NciChannelTan: BLAD StartStop! Kod: %d', UDINT_TO_DINT(fbStartStop.nErrId));
    END_IF
    _Error := TRUE;
    _ErrorId := fbStartStop.nErrId;
    fbStartStop(bStart := FALSE, bStop := FALSE, sNciToPlc := stNciToPlc);
ELSIF fbStartStop.bBusy THEN
    fbStartStop(bStart := FALSE, sNciToPlc := stNciToPlc);
ELSIF NOT fbStartStop.bBusy AND fbStartStop.bStop THEN
    fbStartStop(bStop := FALSE, sNciToPlc := stNciToPlc);
END_IF


IF fbUngroup.bErr THEN
    IF fbUngroup.bExecute THEN
        ADSLOGDINT(ADSLOG_MSGTYPE_ERROR, 'NciChannelTan: BLAD rozpinania grupy! Kod: %d', UDINT_TO_DINT(fbUngroup.nErrId));
    END_IF
    _Error := TRUE;
    _ErrorId := fbUngroup.nErrId;
    fbUngroup(bExecute := FALSE);
    _IsGrouped := FALSE;
ELSIF fbUngroup.bBusy = FALSE AND fbUngroup.bExecute THEN
    ADSLOGSTR(ADSLOG_MSGTYPE_HINT, 'NciChannelTan: Grupa rozpieta pomyslnie.', '');
    _IsGrouped := FALSE;
    fbUngroup(bExecute := FALSE);
END_IF

IF fbBuildExtGroup.bErr THEN
    IF fbBuildExtGroup.bExecute THEN
        ADSLOGDINT(ADSLOG_MSGTYPE_ERROR, 'NciChannelTan: BLAD budowania grupy rozszerzonej! Kod: %d', UDINT_TO_DINT(fbBuildExtGroup.nErrId));
    END_IF
    _Error := TRUE;
    _ErrorId := fbBuildExtGroup.nErrId;
    fbBuildExtGroup(bExecute := FALSE); 
ELSIF fbBuildExtGroup.bBusy = FALSE AND fbBuildExtGroup.bExecute THEN
    ADSLOGSTR(ADSLOG_MSGTYPE_HINT, 'NciChannelTan: Grupa rozszerzona (X,Y,Z,Q) zbudowana pomyslnie.', '');
    _IsGrouped := TRUE;
    fbBuildExtGroup(bExecute := FALSE);
END_IF

IF fbReset.bErr THEN
    _Error := TRUE;
    _ErrorId := fbReset.nErrId;
    fbReset(bExecute := FALSE, sNciToPlc := stNciToPlc);
ELSIF fbReset.bBusy = FALSE AND fbReset.bExecute THEN
    fbReset(bExecute := FALSE, sNciToPlc := stNciToPlc);
END_IF
END_METHOD

PROPERTY IsChannelDone : BOOL
GET
IsChannelDone := _IsChannelDone;
END_GET
END_PROPERTY

PROPERTY IsFeedingDone : BOOL
GET
IsFeedingDone := _IsFeedingDone;
END_GET
END_PROPERTY

PROPERTY IsGrouped : BOOL
GET
IsGrouped := _IsGrouped;
END_GET
END_PROPERTY

PROPERTY IsReady : BOOL
GET
IsReady := (stNciToPlc.ItpState = 2);
END_GET
END_PROPERTY

METHOD ResetChannel
fbStartStop(bStart := FALSE, bStop := FALSE, sNciToPlc := stNciToPlc);

_bResetFeed := TRUE; // <-- ZMIANA: Zamiast lokalnego wywołania, ustawiamy flagę
_bExecuteFeed := FALSE; 

fbReset(
    bExecute := TRUE,
    sNciToPlc := stNciToPlc
);

_Error := FALSE;
_ErrorId := 0;
END_METHOD

METHOD Start
fbStartStop(
    bStart := TRUE, 
    bStop := FALSE,
    sNciToPlc := stNciToPlc 
);
END_METHOD

METHOD StartFeedTable
VAR_IN_OUT
    stTable : ST_NciFeedGroupTable;
END_VAR
// Pobieramy referencję do tabeli (która np. fizycznie leży w Executorze)
refFeedTable REF= stTable;

// Zerujemy flagi gotowości
_IsFeedingDone := FALSE;
_IsChannelDone := FALSE;

// Wyzwalamy blok feedujący
_bExecuteFeed := TRUE;
END_METHOD

METHOD Stop
fbStartStop(
    bStart := FALSE, 
    bStop := TRUE,
    sNciToPlc := stNciToPlc
);
END_METHOD

METHOD Ungroup
fbUngroup(
    bExecute := TRUE, 
    nGroupId := nGroupId
);
END_METHOD

END_FUNCTION_BLOCK

// ---- POUs/Components/FB_Cylinder.TcPOU
FUNCTION_BLOCK FB_Cylinder EXTENDS FB_ComponentBase IMPLEMENTS I_Cylinder
VAR
    
    _ExtendRequest  : BOOL;
    _RetractRequest : BOOL;
    _Extended       : BOOL;
    _Retracted      : BOOL;
    _Extending      : BOOL;
    _Retracting     : BOOL;
	




    Extend_RTRIG  : R_TRIG;
    Retract_RTRIG : R_TRIG;

    //HMI 
    Cylinder_HMI : ST_Cylinder_HMI;
	

    MovementTimer : TON;
    

    CylinderAlarms : ARRAY[1..3] OF FB_TcAlarm;
END_VAR

VAR_INPUT
   	Sensor 			AT%I*		:	BOOL;
END_VAR

VAR_OUTPUT
	Valve			AT%Q*		:	BOOL;
END_VAR

PROPERTY Config : ST_Cylinder_Config
GET
Config := Cylinder_HMI.Config;
END_GET
SET
Cylinder_HMI.Config := Config;
END_SET
END_PROPERTY

METHOD PROTECTED CreateEvents
VAR_INPUT
END_VAR
// Powiązanie tablicy alarmów z klasą CylinderAlarms z TMC
F_CreateAllEventsInClass(
    Alarms     := CylinderAlarms,
    ClassSize  := SIZEOF(TC_EVENTS.CylinderAlarms),
    pInitEvent := ADR(TC_EVENTS.CylinderAlarms.InitReferenceEvent),
    Prefix     := _Name
);


SUPER^.CreateEvents();
END_METHOD

METHOD CyclicLogic
// One shot the requests
Extend_RTRIG(CLK := _ExtendRequest);
Retract_RTRIG(CLK := _RetractRequest);

// Handle Extend
IF Extend_RTRIG.Q THEN
    Valve := TRUE;
    _Extending       := TRUE;
    _Retracting      := FALSE;
    _Retracted       := FALSE;
    _RetractRequest  := FALSE;
END_IF

// Handle Retract
IF Retract_RTRIG.Q THEN
    Valve := FALSE;
    _Extending       := FALSE;
    _Retracting      := TRUE;
    _Extended        := FALSE;
    _ExtendRequest   := FALSE;
END_IF

// Aktualizacja stanu wyłącznie z czujnika
_Extended  := Sensor;
_Retracted := NOT Sensor;

// Status ruchu – tylko gdy trwa przejście
_Extending  := _Extending  AND NOT _Extended;
_Retracting := _Retracting AND NOT _Retracted;

// Odmierzanie czasu ruchu (używamy SEL żeby brać czas wysuwu lub chowania)
MovementTimer(
    IN := _Extending OR _Retracting,
    PT := LREAL_TO_TIME(SEL(_Extending, Cylinder_HMI.Config.RetractTime, Cylinder_HMI.Config.ExtendTime) * 1000.0) 
);

// Wywołanie logiki bazowej komponentu (Tylko raz!)
SUPER^.CyclicLogic();

// Aktualizacja najwyższego priorytetu błędu dla komponentu
_CurrentAlarmSeverity := F_GetMaxSeverityRaised(Alarms := CylinderAlarms, CurrentSeverity := _CurrentAlarmSeverity);
END_METHOD

PROPERTY Error : BOOL
GET
Error := _Error;
END_GET
SET
_Error := Error;
END_SET
END_PROPERTY

METHOD Extend
_ExtendRequest  := TRUE;
_RetractRequest := FALSE;
END_METHOD

PROPERTY Extended : BOOL
GET
Extended := _Extended;
END_GET
END_PROPERTY

METHOD PROTECTED HMICommunication
VAR_INPUT
END_VAR
SUPER^.HMICommunication();

//Handle the requests to extend and retract
IF ComponentBase_HMI.Status.HMIControlAvailable THEN
    IF Cylinder_HMI.Command.Extend THEN
        Extend();
    ELSIF Cylinder_HMI.Command.Retract THEN
        Retract();
    END_IF
END_IF

//Update HMI status info
Cylinder_HMI.Status.Extended    := _Extended;
Cylinder_HMI.Status.Extending   := _Extending;
Cylinder_HMI.Status.Retracted   := _Retracted;
Cylinder_HMI.Status.Retracting  := _Retracting;
END_METHOD

//! @summary Basic component initialization logic
METHOD PROTECTED Initialize : BOOL;

//! @description This method is called by <c>CyclicLogic()</c> as required

IF Sensor THEN
    _Extended  := TRUE;
    _Retracted := FALSE;
ELSE
    _Extended  := FALSE;
    _Retracted := TRUE;
END_IF

_Extending      := FALSE;
_ExtendRequest  := FALSE;
_Retracting     := FALSE;
_RetractRequest := FALSE;

Initialize := SUPER^.Initialize();
END_METHOD

METHOD PROTECTED Monitoring
VAR_INPUT
END_VAR
_Busy := _Extending OR _Retracting;

// Jeśli czas minął, zgłoś odpowiedni błąd
IF MovementTimer.Q THEN
    _Error   := TRUE;
    _ErrorID := 1; 


    IF _Extending AND NOT CylinderAlarms[E_CylinderAlarms.ExtendTimeout].bRaised THEN
        RaiseAlarmWithStrings(CylinderAlarms[E_CylinderAlarms.ExtendTimeout], '', '');
    
    ELSIF _Retracting AND NOT CylinderAlarms[E_CylinderAlarms.RetractTimeout].bRaised THEN
        RaiseAlarmWithStrings(CylinderAlarms[E_CylinderAlarms.RetractTimeout], '', '');
    END_IF
END_IF

// Resetowanie błędu i ALARMÓW, gdy cylinder w końcu dotrze do celu
IF (_Extended AND _ExtendRequest) OR (_Retracted AND _RetractRequest) THEN
    _Error   := FALSE;
    _ErrorID := 0;
    
    // Musimy zdjąć alarmy, żeby system bazowy nie podniósł flagi błędu ponownie!
    CylinderAlarms[E_CylinderAlarms.ExtendTimeout].Clear(0,0);
    CylinderAlarms[E_CylinderAlarms.RetractTimeout].Clear(0,0);
END_IF

SUPER^.Monitoring();
END_METHOD

METHOD Retract
_ExtendRequest  := FALSE;
_RetractRequest := TRUE;
END_METHOD

PROPERTY Retracted : BOOL
GET
Retracted := _Retracted;
END_GET
END_PROPERTY

END_FUNCTION_BLOCK

// ---- POUs/GantryXYZ/HomingStrategies/FB_Homing_StandardNC.TcPOU
FUNCTION_BLOCK FB_Homing_StandardNC EXTENDS FB_Homing_Base IMPLEMENTS I_MotionSequence
VAR
    fbMcHome           : MC_Home;
    fbMoveAbs          : MC_MoveAbsolute;
    _ReferencePosition : LREAL;	
    _RapidVelocity     : LREAL := 100.0; 
	_HomingVelocity	   : LREAL := 10.0;
END_VAR
VAR_INPUT
    bSensorInput : BOOL;
	bForceHoming : BOOL := FALSE;
END_VAR

METHOD Abort
VAR_INPUT
END_VAR
fbMcHome(Axis := _Axis.Axis, Execute := FALSE);
fbMoveAbs(Axis := _Axis.Axis, Execute := FALSE);
_bBusy := FALSE;
nStep := 0;
END_METHOD

METHOD CyclicLogic
CASE nStep OF
    0: 
        fbMcHome(Axis := _Axis.Axis, Execute := FALSE);
        fbMoveAbs(Axis := _Axis.Axis, Execute := FALSE);

	10: 
        IF _Axis.Axis.Status.Homed AND NOT bForceHoming THEN
            nStep := 15; 
        ELSE
            nStep := 20; 
        END_IF

    15: 
        fbMoveAbs(
            Axis     := _Axis.Axis,
            Execute  := TRUE,
            Position := _ReferencePosition,
            Velocity := _RapidVelocity 
        );
        
        IF fbMoveAbs.Done THEN
            fbMoveAbs(Axis := _Axis.Axis, Execute := FALSE); 
            
            _bBusy := FALSE;
            _bDone := TRUE;
            nStep  := 0; 
            
        ELSIF fbMoveAbs.Error THEN
            nStep := 99;
        END_IF

    20: 
        fbMcHome(
            Axis            := _Axis.Axis, 
            Execute         := TRUE, 
            HomingMode      := MC_DefaultHoming,
            bCalibrationCam := bSensorInput
        );
        
        IF fbMcHome.Busy THEN
            nStep := 25;
        ELSIF fbMcHome.Error THEN
            nStep := 99;
        END_IF

	25: 
        fbMcHome(
            Axis            := _Axis.Axis,
            bCalibrationCam := bSensorInput 
        );
        IF fbMcHome.Done THEN
            fbMcHome(Axis := _Axis.Axis, Execute := FALSE);
            nStep := 26; 
        ELSIF fbMcHome.Error THEN
            nStep := 99;
        END_IF

    26:
        
        IF NOT fbMcHome.Busy AND _Axis.Axis.Status.StandStill THEN
            nStep := 30;
        END_IF

    30: 
        fbMoveAbs(
            Axis     := _Axis.Axis,
            Execute  := TRUE,
            Position := _ReferencePosition,
            Velocity := _HomingVelocity
        );
		
		IF NOT fbMoveAbs.Busy AND _Axis.Axis.Status.StandStill THEN
			nStep := 32;
		END_IF
	
	32:	
        
        IF fbMoveAbs.Done THEN
            fbMoveAbs(Axis := _Axis.Axis, Execute := FALSE);
            _bBusy := FALSE;
            _bDone := TRUE;
            nStep  := 0;
        ELSIF fbMoveAbs.Error THEN
            nStep := 99;
        END_IF

    99: 
        _bBusy    := FALSE;
        _bError   := TRUE;
        
        IF fbMoveAbs.Error THEN
            _bErrorID := fbMoveAbs.ErrorID;
        ELSE
            _bErrorID := fbMcHome.ErrorID;
        END_IF
        
        nStep     := 0;
END_CASE
END_METHOD

PROPERTY HomingVelocity : LREAL
GET
HomingVelocity := _HomingVelocity;
END_GET
SET
_HomingVelocity := HomingVelocity;
END_SET
END_PROPERTY

PROPERTY RapidVelocity : LREAL
GET
RapidVelocity := _RapidVelocity;
END_GET
SET
_RapidVelocity := RapidVelocity;
END_SET
END_PROPERTY

PROPERTY ReferencePosition : LREAL
GET
ReferencePosition := _ReferencePosition;
END_GET
SET
_ReferencePosition := ReferencePosition;
END_SET
END_PROPERTY

END_FUNCTION_BLOCK

// ---- POUs/GantryXYZ/HomingStrategies/FB_Homing_Base.TcPOU
FUNCTION_BLOCK FB_Homing_Base EXTENDS FB_CyclicFB IMPLEMENTS I_HomingStrategy
VAR
    _Axis     : SPT_Motion_Control.I_BasicAxis;
    _bBusy    : BOOL;
    _bDone    : BOOL;
    _bError   : BOOL;
    _bErrorID : UDINT;
    nStep     : INT;
END_VAR

METHOD Abort
VAR_INPUT
END_VAR
_bBusy := FALSE;
nStep := 0;
END_METHOD

PROPERTY Axis : SPT_Motion_Control.I_BasicAxis
GET
Axis := _Axis;
END_GET
SET
_Axis := Axis;
END_SET
END_PROPERTY

PROPERTY Busy : BOOL
GET
Busy := _bBusy;
END_GET
END_PROPERTY

METHOD CyclicLogic
// Pusta metoda w klasie bazowej - musi być nadpisana przez dzieci!
END_METHOD

PROPERTY Done : BOOL
GET
Done := _bDone;
END_GET
END_PROPERTY

PROPERTY Error : BOOL
GET
Error := _bError;
END_GET
END_PROPERTY

PROPERTY ErrorID : UDINT
GET
ErrorID := _bErrorID;
END_GET
END_PROPERTY

METHOD Execute : BOOL
IF _Axis = 0 THEN RETURN; END_IF

_bBusy       := TRUE;
_bDone       := FALSE;
_bError      := FALSE;
_bErrorID    := 0;
nStep        := 10; // Start sekwencji
Execute      := TRUE;
END_METHOD

PROPERTY InitComplete : BOOL
GET
InitComplete := TRUE;
END_GET
END_PROPERTY

END_FUNCTION_BLOCK

// ---- POUs/GantryXYZ/HomingStrategies/FB_Homing_Direct.TcPOU
FUNCTION_BLOCK FB_Homing_Direct EXTENDS FB_Homing_Base
VAR_INPUT
    ReferencePosition : LREAL := 0.0;
END_VAR
VAR
    fbMcHome          : MC_Home;
    fbMoveAbs         : MC_MoveAbsolute;
    DelayTimer        : TON;
	_HomingVelocity   : LREAL := 50.0;
END_VAR

METHOD Abort
VAR_INPUT
END_VAR
IF _Axis <> 0 THEN
    fbMcHome(Axis := _Axis.Axis, Execute := FALSE);
    fbMoveAbs(Axis := _Axis.Axis, Execute := FALSE);
END_IF

SUPER^.Abort();
END_METHOD

METHOD CyclicLogic
CASE nStep OF
    0: 
        fbMcHome(Axis := _Axis.Axis, Execute := FALSE);
        fbMoveAbs(Axis := _Axis.Axis, Execute := FALSE);

    10: 
        IF _Axis.Axis.Status.Homed THEN
            nStep := 20;
        ELSE
            fbMcHome(
                Axis        := _Axis.Axis, 
                Execute     := TRUE, 
                Position    := ReferencePosition,
                HomingMode  := MC_Direct
            );
            
            IF fbMcHome.Done THEN
                fbMcHome(Axis := _Axis.Axis, Execute := FALSE);
                nStep := 20;
            ELSIF fbMcHome.Error THEN
                _bBusy    := FALSE;
                _bError   := TRUE;
                _bErrorID := fbMcHome.ErrorID;
                nStep     := 0;
            END_IF
        END_IF

    20: 
        fbMoveAbs(
            Axis     := _Axis.Axis,
            Execute  := TRUE,
			Velocity := _HomingVelocity,
            Position := 0.0
        );
        
        IF fbMoveAbs.Done THEN
            fbMoveAbs(Axis := _Axis.Axis, Execute := FALSE);
            nStep := 40;
        ELSIF fbMoveAbs.Error THEN
            _bBusy    := FALSE;
            _bError   := TRUE;
            _bErrorID := fbMoveAbs.ErrorID;
            nStep     := 0;
        END_IF
        
    40: 
        _bBusy := FALSE;
        _bDone := TRUE; 
        nStep  := 0;
END_CASE
END_METHOD

PROPERTY HomingVelocity : LREAL
GET
HomingVelocity := _HomingVelocity;
END_GET
SET
_HomingVelocity := HomingVelocity;
END_SET
END_PROPERTY

END_FUNCTION_BLOCK

// ---- POUs/FB_PersistentDataManager.TcPOU
FUNCTION_BLOCK FB_PersistentDataManager
VAR PERSISTENT
    _PanelFrontLength : REAL;
    _Config           : ST_RecipeBuilder_Config;
    _GantryConfig     : ST_GantryXYZ_Config; 
END_VAR

PROPERTY Config : ST_RecipeBuilder_Config
GET
Config := _Config;
END_GET
SET
_Config := Config;
END_SET
END_PROPERTY

PROPERTY GantryConfig : ST_GantryXYZ_Config
GET
GantryConfig := _GantryConfig;
END_GET
SET
_GantryConfig := GantryConfig;
END_SET
END_PROPERTY

END_FUNCTION_BLOCK

// ---- POUs/Builder/FB_RecipeFactory.TcPOU
FUNCTION_BLOCK FB_RecipeFactory
VAR
    BuilderWings 			: FB_PTPBorgoWings;
    BuilderFlaps 			: FB_PTPBorgoFlaps;
    BuilderArona 			: FB_PTPArona;
	BuilderRectangle 		: FB_PTPRectangle;
	
	BuilderCircle 			: FB_NCICircle;
	
	BuilderRoundedRect 		: FB_FeedRoundedRectangle;	
	BuilderFeedCircle  		: FB_FeedCircle;
	
	BuilderMeina2_2000x1000				: FB_FeedMeina2_2000x1000;
	BuilderMeina2_5Squares    			: FB_FeedMeina2_500x500;
    BuilderMeina2_500x500_Circles    	: FB_FeedMeina2_500x500_Circles;
    BuilderMeina2_3Squares    			: FB_FeedMeina2_750x750;
    BuilderMeina2_3Circles    			: FB_FeedMeina2_750x750_Circles;
    BuilderMeina2_1000x1000   			: FB_FeedMeina2_1000x1000;
    BuilderMeina2_1000x1000_Circles    	: FB_FeedMeina2_1000x1000_Circles;
    BuilderMeina2_2000x500    			: FB_FeedMeina2_2000x500;
	
	BuilderMeina2_Samples				: FB_FeedMeina2_Samples;
END_VAR

METHOD GetBuilder : I_RecipeBuilder
VAR_INPUT
    RequestedRecipe : E_RecipeID;
END_VAR
CASE RequestedRecipe OF
    E_RecipeID.ePTPBorgoWings:
        GetBuilder := BuilderWings; 
        
    E_RecipeID.ePTPBorgoFlaps:
        GetBuilder := BuilderFlaps;
        
    E_RecipeID.ePTPArona:
        GetBuilder := BuilderArona;
		
	E_RecipeID.eNCICircle:
        GetBuilder := BuilderCircle;
		
	E_RecipeID.ePTPRectangle:                            
        GetBuilder := BuilderRectangle; 
	
	E_RecipeID.eFeedRoundedRectangle:                            
        GetBuilder := BuilderRoundedRect;    

	E_RecipeID.eFeedCircle:                 
        GetBuilder := BuilderFeedCircle;        

	E_RecipeID.eFeedMeina2_2000x1000:
		GetBuilder := BuilderMeina2_2000x1000;   
		
	E_RecipeID.eFeedMeina2_500x500:    
		GetBuilder := BuilderMeina2_5Squares;
		
    E_RecipeID.eFeedMeina2_500x500_Circles:    
		GetBuilder := BuilderMeina2_500x500_Circles;
		
    E_RecipeID.eFeedMeina2_750x750:    
		GetBuilder := BuilderMeina2_3Squares;
		
    E_RecipeID.eFeedMeina2_750x750_Circles:    
		GetBuilder := BuilderMeina2_3Circles;
		
    E_RecipeID.eFeedMeina2_1000x1000:    
		GetBuilder := BuilderMeina2_1000x1000;
		
    E_RecipeID.eFeedMeina2_1000x1000_Circles:    
		GetBuilder := BuilderMeina2_1000x1000_Circles;
		
    E_RecipeID.eFeedMeina2_2000x500: 
		GetBuilder := BuilderMeina2_2000x500;
		
	E_RecipeID.eFeedMeina2_Samples: 
		GetBuilder := BuilderMeina2_Samples;	
        
ELSE
    GetBuilder := 0; 
END_CASE
END_METHOD

METHOD InitializeFactory
VAR_INPUT
    Config : ST_RecipeBuilder_Config;
	ConfigProvider : I_GantryConfigProvider;
END_VAR
BuilderWings.Config 				:= Config;
BuilderWings.ConfigProvider 		:= ConfigProvider; 

BuilderFlaps.Config 				:= Config;
BuilderFlaps.ConfigProvider 		:= ConfigProvider;

BuilderArona.Config 				:= Config;
BuilderArona.ConfigProvider 		:= ConfigProvider;

BuilderCircle.Config 				:= Config;
BuilderCircle.ConfigProvider 		:= ConfigProvider;

BuilderRectangle.Config 			:= Config;                    
BuilderRectangle.ConfigProvider 	:= ConfigProvider; 
   
BuilderRoundedRect.Config 			:= Config;
BuilderRoundedRect.ConfigProvider 	:= ConfigProvider;

BuilderFeedCircle.Config 			:= Config;                    
BuilderFeedCircle.ConfigProvider 	:= ConfigProvider;

BuilderMeina2_2000x1000.Config				:= Config;    
BuilderMeina2_2000x1000.ConfigProvider		:= ConfigProvider;

BuilderMeina2_5Squares.Config       := Config;
BuilderMeina2_5Squares.ConfigProvider := ConfigProvider;

BuilderMeina2_500x500_Circles.Config       := Config;
BuilderMeina2_500x500_Circles.ConfigProvider := ConfigProvider;

BuilderMeina2_3Squares.Config       := Config;
BuilderMeina2_3Squares.ConfigProvider := ConfigProvider;

BuilderMeina2_3Circles.Config       := Config;
BuilderMeina2_3Circles.ConfigProvider := ConfigProvider;

BuilderMeina2_1000x1000.Config       := Config;
BuilderMeina2_1000x1000.ConfigProvider := ConfigProvider;

BuilderMeina2_1000x1000_Circles.Config       := Config;
BuilderMeina2_1000x1000_Circles.ConfigProvider := ConfigProvider;

BuilderMeina2_2000x500.Config    := Config;
BuilderMeina2_2000x500.ConfigProvider := ConfigProvider;    

BuilderMeina2_Samples.Config    := Config;
BuilderMeina2_Samples.ConfigProvider := ConfigProvider;
END_METHOD

METHOD UpdateConfig
VAR_INPUT
    Config : ST_RecipeBuilder_Config;
END_VAR
// Fabryka rozsyła nową konfigurację do wszystkich swoich "dzieci"
BuilderWings.Config 		:= Config;
BuilderFlaps.Config 		:= Config;
BuilderArona.Config 		:= Config;
BuilderCircle.Config 		:= Config;
BuilderRectangle.Config 	:= Config;   
BuilderRoundedRect.Config 	:= Config;      
BuilderFeedCircle.Config 	:= Config; 
BuilderMeina2_2000x1000.Config		:= Config;                 
BuilderMeina2_5Squares.Config    := Config;
BuilderMeina2_500x500_Circles.Config    := Config;
BuilderMeina2_3Squares.Config    := Config;
BuilderMeina2_3Circles.Config    := Config;
BuilderMeina2_1000x1000.Config    := Config;
BuilderMeina2_1000x1000_Circles.Config    := Config;
BuilderMeina2_2000x500.Config := Config;
BuilderMeina2_Samples.Config := Config;
END_METHOD

END_FUNCTION_BLOCK

// ---- POUs/Builder/Recipes/FB_PTPBorgoWings.TcPOU
FUNCTION_BLOCK FB_PTPBorgoWings EXTENDS FB_RecipeBase

METHOD Build : BOOL
VAR_INST
    TotalY          : REAL;
    TotalX          : REAL;
    ShorterY        : REAL;
    ShorterX        : REAL;
END_VAR
_Busy := TRUE;
_Done := FALSE;
_Error := FALSE;
Build := FALSE;

THIS^.UpdateNestingLimits();

// 2. Jeśli detal wystaje poza maszynę - przerywamy od razu!
IF NOT _Config.IsValid THEN
    _Busy := FALSE;
    _Error := TRUE; 
    Build := FALSE;
    RETURN;
END_IF

// 3. Pobieramy wyliczone gabaryty nominalne do lokalnych zmiennych roboczych
TotalX   := _NominalX;
TotalY   := _NominalY; 
ShorterY := TotalY - _Config.PanelHeight;
ShorterX := TotalX - _Config.PanelHeight;


// ------------------------------------
// 1. Segregracja frezowania (Grooving)
// ------------------------------------
_SegmentsToGroove := 4;

_SegmentsGroove[1].Start.X := TotalX;
_SegmentsGroove[1].Stop.X  := 0;
_SegmentsGroove[1].Start.Y := ShorterY;
_SegmentsGroove[1].Stop.Y  := ShorterY;

_SegmentsGroove[2].Start.X := TotalX;
_SegmentsGroove[2].Stop.X  := 0; 
_SegmentsGroove[2].Start.Y := _Config.PanelHeight;
_SegmentsGroove[2].Stop.Y  := _Config.PanelHeight;

_SegmentsGroove[3].Start.X := ShorterX;
_SegmentsGroove[3].Stop.X  := ShorterX;
_SegmentsGroove[3].Start.Y := TotalY;
_SegmentsGroove[3].Stop.Y  := 0;

_SegmentsGroove[4].Start.Y := TotalY;
_SegmentsGroove[4].Stop.Y  := 0;
_SegmentsGroove[4].Start.X := _Config.PanelHeight;
_SegmentsGroove[4].Stop.X  := _Config.PanelHeight;

// ------------------------------------
// 2. Cięcie w osi X (Cut X)
// ------------------------------------
_SegmentsToCutX := 6;

// Short Box Segments
_SegmentsCutX[1].Start.X := TotalX + _Config.CuttingOverpass;
_SegmentsCutX[1].Stop.X  := ShorterX;
_SegmentsCutX[1].Start.Y := ShorterY;
_SegmentsCutX[1].Stop.Y  := ShorterY;

_SegmentsCutX[2].Start.X := _Config.PanelHeight;
_SegmentsCutX[2].Stop.X  := -_Config.CuttingOverpass;
_SegmentsCutX[2].Start.Y := ShorterY;
_SegmentsCutX[2].Stop.Y  := ShorterY;

_SegmentsCutX[3].Start.X := TotalX + _Config.CuttingOverpass;
_SegmentsCutX[3].Stop.X  := ShorterX;
_SegmentsCutX[3].Start.Y := _Config.PanelHeight;
_SegmentsCutX[3].Stop.Y  := _Config.PanelHeight;

_SegmentsCutX[4].Start.X := _Config.PanelHeight;
_SegmentsCutX[4].Stop.X  := -_Config.CuttingOverpass;
_SegmentsCutX[4].Start.Y := _Config.PanelHeight;
_SegmentsCutX[4].Stop.Y  := _Config.PanelHeight;

// Panel Dimensions Shorter Flaps
_SegmentsCutX[5].Start.X := TotalX + _Config.CuttingOverpass;
_SegmentsCutX[5].Stop.X  := -_Config.CuttingOverpass;
_SegmentsCutX[5].Start.Y := TotalY - _Config.RailHeightCorrection;
_SegmentsCutX[5].Stop.Y  := TotalY - _Config.RailHeightCorrection;

_SegmentsCutX[6].Start.X := TotalX + _Config.CuttingOverpass;
_SegmentsCutX[6].Stop.X  := -_Config.CuttingOverpass;
_SegmentsCutX[6].Start.Y := _Config.RailHeightCorrection;
_SegmentsCutX[6].Stop.Y  := _Config.RailHeightCorrection;

// ------------------------------------
// 3. Cięcie w osi Y (Cut Y)
// ------------------------------------
_SegmentsToCutY := 6;

// Short Box Segments
_SegmentsCutY[1].Start.X := ShorterX;
_SegmentsCutY[1].Stop.X  := ShorterX;
_SegmentsCutY[1].Start.Y := TotalY + _Config.CuttingOverpass;
_SegmentsCutY[1].Stop.Y  := ShorterY;

_SegmentsCutY[2].Start.X := _Config.PanelHeight;
_SegmentsCutY[2].Stop.X  := _Config.PanelHeight;
_SegmentsCutY[2].Start.Y := TotalY + _Config.CuttingOverpass;
_SegmentsCutY[2].Stop.Y  := ShorterY;

_SegmentsCutY[3].Start.X := ShorterX;
_SegmentsCutY[3].Stop.X  := ShorterX;
_SegmentsCutY[3].Start.Y := _Config.PanelHeight;
_SegmentsCutY[3].Stop.Y  := -_Config.CuttingOverpass;

_SegmentsCutY[4].Start.X := _Config.PanelHeight;
_SegmentsCutY[4].Stop.X  := _Config.PanelHeight;
_SegmentsCutY[4].Start.Y := _Config.PanelHeight;
_SegmentsCutY[4].Stop.Y  := -_Config.CuttingOverpass;

// Panel Dimensions
_SegmentsCutY[5].Start.X := TotalX;
_SegmentsCutY[5].Stop.X  := TotalX;
_SegmentsCutY[5].Start.Y := TotalY + _Config.CuttingOverpass;
_SegmentsCutY[5].Stop.Y  := -_Config.CuttingOverpass;

_SegmentsCutY[6].Start.X := 0;
_SegmentsCutY[6].Stop.X  := 0;
_SegmentsCutY[6].Start.Y := TotalY + _Config.CuttingOverpass;
_SegmentsCutY[6].Stop.Y  := -_Config.CuttingOverpass;


_Busy := FALSE;
_Done := TRUE;
Build := TRUE;
END_METHOD

METHOD PROTECTED CalculateFootprint
VAR_INPUT
END_VAR
// BorgoWings wie, że jego wymiar powiększa się o ścianki zagięcia:
_NominalX := _Config.PanelFrontWidth  + 2.0 * _Config.PanelHeight;
_NominalY := _Config.PanelFrontLength + 2.0 * _Config.PanelHeight;
END_METHOD

PROPERTY ExecutionRoute : E_ExecutionRoute
GET
ExecutionRoute := E_ExecutionRoute.ePTP;
END_GET
END_PROPERTY

METHOD FB_init : BOOL
VAR_INPUT
	bInitRetains : BOOL; // if TRUE, the retain variables are initialized (warm start / cold start)
	bInCopyCode : BOOL;  // if TRUE, the instance afterwards gets moved into the copy code (online change)
END_VAR
_Limits.PanelFrontLength.MinVal := 100.0;
_Limits.PanelFrontLength.MaxVal := 1234.0;

_Limits.PanelFrontWidth.MinVal  := 100.0;
_Limits.PanelFrontWidth.MaxVal  := 1234.0;

_Limits.PanelHeight.MinVal      := 0.0;
_Limits.PanelHeight.MaxVal      := 1234.0;

_Limits.RailHeightCorrection.MinVal := 12.0;
_Limits.RailHeightCorrection.MaxVal := 14.0;

_Limits.CuttingOverpass.MinVal := 0.0;
_Limits.CuttingOverpass.MaxVal := 50.0;

_Limits.GroovingOverpass.MinVal := 0.0;
_Limits.GroovingOverpass.MaxVal := 50.0;

_Limits.GrooveDepthZ.MinVal := 0.0;
_Limits.GrooveDepthZ.MaxVal := 9.0; //
END_METHOD

END_FUNCTION_BLOCK

// ---- POUs/Builder/FB_RecipeBase.TcPOU
FUNCTION_BLOCK FB_RecipeBase IMPLEMENTS I_RecipeBuilder 

VAR
    _Config                 : ST_RecipeBuilder_Config;
	_ConfigProvider 		: I_GantryConfigProvider;

	
	
	_Limits : ST_Recipe_Limits;

    // --- NOWE ZMIENNE DO PRZECHOWYWANIA SEGMENTÓW ---
    _SegmentsCutX           : ARRAY [1..100] OF ST_CutSegment;
    _SegmentsCutY           : ARRAY [1..100] OF ST_CutSegment;
    _SegmentsGroove         : ARRAY [1..100] OF ST_CutSegment;
	_HolesDrill 			: ARRAY [1..100] OF ST_PointXY;
	_ShapeStart         	: ARRAY [1..100] OF ST_PointXY;
	_ShapesCount        	: INT := 1;
    _CurrentShapeIndex  	: INT := 1;
	_HolesToDrill   		: INT;
    _SegmentsToCutX         : INT;
    _SegmentsToCutY         : INT;
    _SegmentsToGroove       : INT;
	_FootprintX 			: REAL;
	_FootprintY 			: REAL;
	_MaxCopiesX				: DINT;
	_MaxCopiesY				: DINT;
	_ActualCopiesX			: DINT;
	_ActualCopiesY			: DINT;
	_NominalX 				: REAL;
    _NominalY 				: REAL;
	_Busy					: BOOL;
	_Done					: BOOL;
	_Error					: BOOL;
	
	// --- GENERYCZNY GENERATOR G-CODE (NCI) ---
    fbCreateFile    : ItpPpgCreateMain;
    fbAppendLine    : ItpPpgAppendGenericBlock;
    fbCloseFile     : ItpPpgCloseMain;
    
    _aGCodeBuffer   : ARRAY[1..600] OF STRING(255); 
    _nLinesToWrite  : INT;                          // Ile linii z bufora zapisać
    _nFileWriteStep : INT := 0;                     // Krok maszyny stanów zapisu
    _sGCodeFilePath : STRING(255);                  // Ścieżka pliku
	
	_GeometryWriter : I_GeometryWriter;
	
END_VAR

PROPERTY ActualCopiesX : DINT
GET
ActualCopiesX := _Config.RequestedCopiesX;
END_GET
END_PROPERTY

PROPERTY ActualCopiesY : DINT
GET
ActualCopiesY := _Config.RequestedCopiesY;
END_GET
END_PROPERTY

METHOD Build : BOOL
Build := FALSE;
END_METHOD

PROPERTY Busy : BOOL
GET
Busy := _Busy;
END_GET
SET
_Busy := Busy;
END_SET
END_PROPERTY

METHOD PROTECTED CalculateFootprint
VAR_INPUT
END_VAR
// Domyślny wymiar detalu (bez dodatków)
_NominalX := _Config.PanelFrontWidth;
_NominalY := _Config.PanelFrontLength;
END_METHOD

PROPERTY Config : ST_RecipeBuilder_Config
GET
Config := _Config;
END_GET
SET
VAR
    sTempGCodePath : STRING(255);
END_VAR
// 1. NAJPIERW robimy kopię tego co mamy w pamięci sterownika
sTempGCodePath := THIS^._Config.GCodePath; 

// 2. TERAZ przyjmujemy nową strukturę z HMI
_Config := Config;

// 3. PRZYWRACAMY ścieżkę do pliku
_Config.GCodePath := sTempGCodePath;

_Config.PanelFrontLength     := LIMIT(_Limits.PanelFrontLength.MinVal, Config.PanelFrontLength, _Limits.PanelFrontLength.MaxVal);
_Config.PanelFrontWidth      := LIMIT(_Limits.PanelFrontWidth.MinVal,  Config.PanelFrontWidth,  _Limits.PanelFrontWidth.MaxVal);
_Config.PanelHeight          := LIMIT(_Limits.PanelHeight.MinVal,      Config.PanelHeight,      _Limits.PanelHeight.MaxVal);
_Config.RailHeightCorrection := LIMIT(_Limits.RailHeightCorrection.MinVal, Config.RailHeightCorrection, _Limits.RailHeightCorrection.MaxVal);
_Config.GrooveDepthZ		 :=	LIMIT(_Limits.GrooveDepthZ.MinVal,	Config.GrooveDepthZ, _Limits.GrooveDepthZ.MaxVal);
_Config.Diameter 			 := LIMIT(_Limits.Diameter.MinVal, Config.Diameter, _Limits.Diameter.MaxVal);

_Config.CuttingOverpass      := LIMIT(_Limits.CuttingOverpass.MinVal, Config.CuttingOverpass, _Limits.CuttingOverpass.MaxVal);
_Config.GroovingOverpass     := LIMIT(_Limits.GroovingOverpass.MinVal, Config.GroovingOverpass, _Limits.GroovingOverpass.MaxVal);
_Config.Radius               := LIMIT(_Limits.Radius.MinVal, Config.Radius, _Limits.Radius.MaxVal);

THIS^.UpdateNestingLimits();


IF _Config.FillAll THEN
    _Config.RequestedCopiesX := _MaxCopiesX;
    _Config.RequestedCopiesY := _MaxCopiesY;
ELSE
    _Config.RequestedCopiesX := LIMIT(1, _Config.RequestedCopiesX, _MaxCopiesX);
    _Config.RequestedCopiesY := LIMIT(1, _Config.RequestedCopiesY, _MaxCopiesY);
END_IF
END_SET
END_PROPERTY

PROPERTY ConfigProvider : I_GantryConfigProvider
GET
ConfigProvider := _ConfigProvider;
END_GET
SET
_ConfigProvider := ConfigProvider;
END_SET
END_PROPERTY

PROPERTY CurrentShapeIndex : INT
GET
CurrentShapeIndex := _CurrentShapeIndex;
END_GET
SET
_CurrentShapeIndex := CurrentShapeIndex;
END_SET
END_PROPERTY

PROPERTY Done : BOOL
GET
Done := _Done;
END_GET
SET
_Done := Done;
END_SET
END_PROPERTY

PROPERTY Error : BOOL
GET
Error := _Error;
END_GET
SET
_Error := Error;
END_SET
END_PROPERTY

PROPERTY ExecutionRoute : E_ExecutionRoute
GET
END_GET
END_PROPERTY

PROPERTY FootprintX : REAL
GET
FootprintX := _FootprintX;
END_GET
SET
_FootprintX := FootprintX;
END_SET
END_PROPERTY

PROPERTY FootprintY : REAL
GET
FootprintY := _FootprintY;
END_GET
SET
_FootprintY := FootprintY;
END_SET
END_PROPERTY

PROPERTY GeometryWriter : I_GeometryWriter
GET
GeometryWriter := _GeometryWriter;
END_GET
SET
_GeometryWriter := GeometryWriter;
END_SET
END_PROPERTY

PROPERTY HolesDrill : REFERENCE TO ARRAY [1..100] OF ST_PointXY
GET
HolesDrill REF= _HolesDrill;
END_GET
END_PROPERTY

PROPERTY HolesToDrill : INT
GET
HolesToDrill := _HolesToDrill;
END_GET
END_PROPERTY

PROPERTY Limits : ST_Recipe_Limits
GET
Limits := _Limits;
END_GET
END_PROPERTY

PROPERTY MaxCopiesX : DINT
GET
MaxCopiesX := _MaxCopiesX;
END_GET
END_PROPERTY

PROPERTY MaxCopiesY : DINT
GET
MaxCopiesY := _MaxCopiesY ;
END_GET
END_PROPERTY

PROPERTY SegmentsCutX : REFERENCE TO ARRAY [1..100] OF ST_CutSegment
GET
SegmentsCutX REF= _SegmentsCutX;
END_GET
END_PROPERTY

PROPERTY SegmentsCutY : REFERENCE TO ARRAY [1..100] OF ST_CutSegment
GET
SegmentsCutY REF= _SegmentsCutY;
END_GET
END_PROPERTY

PROPERTY SegmentsGroove : REFERENCE TO ARRAY [1..100] OF ST_CutSegment
GET
SegmentsGroove REF= _SegmentsGroove;
END_GET
END_PROPERTY


PROPERTY SegmentsToCutX : INT
GET
SegmentsToCutX := _SegmentsToCutX;
END_GET
END_PROPERTY


PROPERTY SegmentsToCutY : INT
GET
SegmentsToCutY := _SegmentsToCutY;
END_GET
END_PROPERTY


PROPERTY SegmentsToGroove : INT
GET
SegmentsToGroove := _SegmentsToGroove;
END_GET
END_PROPERTY

PROPERTY ShapesCount : INT
GET
ShapesCount := _ShapesCount;
END_GET
END_PROPERTY

PROPERTY ShapeStart : REFERENCE TO ARRAY [1..100] OF ST_PointXY
GET
ShapeStart REF= _ShapeStart;
END_GET
END_PROPERTY

METHOD PUBLIC UpdateNestingLimits
VAR
    MaxOverpass     : REAL;
    MachineConfig   : ST_GantryXYZ_Config; // Zmienna do odczytu offsetu
    EffectiveBoardX : REAL;
    EffectiveBoardY : REAL;
END_VAR
VAR_INST
    bLogFired       : BOOL; // <-- Zapamięta, czy log już poszedł
END_VAR
// 1. Czysty gabaryt z logiki receptury
THIS^.CalculateFootprint();
MaxOverpass := MAX(_Config.CuttingOverpass, _Config.GroovingOverpass);
_FootprintX := _NominalX + (2.0 * MaxOverpass);
_FootprintY := _NominalY + (2.0 * MaxOverpass);

// 2. Pobranie Global Offsetu ORAZ wymiarów płyty z maszyny
IF _ConfigProvider <> 0 THEN
    MachineConfig := _ConfigProvider.Config;
ELSE
    // Awaryjny "fallback" jeśli Provider nie jest wstrzyknięty (np. w starych testach)
    MachineConfig.GlobalOffsetX := 0.0;
    MachineConfig.GlobalOffsetY := 0.0;
    MachineConfig.RawBoardX := 1220.0; // Domyślna płyta 
    MachineConfig.RawBoardY := 2440.0; // Domyślna płyta
	MachineConfig.RawBoardZ := 9.0;
END_IF

// 3. Efektywna wielkość płyty = Fizyczna płyta (z maszyny) minus offset początkowy
EffectiveBoardX := MachineConfig.RawBoardX - MachineConfig.GlobalOffsetX;
EffectiveBoardY := MachineConfig.RawBoardY - MachineConfig.GlobalOffsetY;

// 4. Przeliczanie kopii nestingu (zabezpieczenie na ujemne wymiary)
IF _FootprintX > 0.0 AND EffectiveBoardX > 0.0 THEN
    _MaxCopiesX := REAL_TO_DINT(TRUNC(EffectiveBoardX / _FootprintX));
ELSE
    _MaxCopiesX := 0;
END_IF

IF _FootprintY > 0.0 AND EffectiveBoardY > 0.0 THEN
    _MaxCopiesY := REAL_TO_DINT(TRUNC(EffectiveBoardY / _FootprintY));
ELSE
    _MaxCopiesY := 0;
END_IF

// =========================================================
// 5. WERYFIKACJA GABARYTÓW (Zabezpieczenie przed za dużym detalem)
// =========================================================
_Config.IsValid := (_MaxCopiesX > 0) AND (_MaxCopiesY > 0) AND (_NominalX > 0) AND (_NominalY > 0);

IF NOT _Config.IsValid THEN
    IF NOT bLogFired THEN
        ADSLOGSTR(ADSLOG_MSGTYPE_ERROR, 'UpdateNestingLimits: Konfiguracja odrzucona (IsValid = FALSE)! Sprawdzam dlaczego...', '');
        
        IF _MaxCopiesX <= 0 THEN 
            ADSLOGSTR(ADSLOG_MSGTYPE_ERROR, 'Powod: _MaxCopiesX <= 0 (Detal wychodzi poza szerokosc stolu)', ''); 
        END_IF
        IF _MaxCopiesY <= 0 THEN 
            ADSLOGSTR(ADSLOG_MSGTYPE_ERROR, 'Powod: _MaxCopiesY <= 0 (Detal wychodzi poza dlugosc stolu)', ''); 
        END_IF
        IF _NominalX <= 0 THEN 
            ADSLOGSTR(ADSLOG_MSGTYPE_ERROR, 'Powod: _NominalX <= 0 (Szerokosc Nominalna to zero!)', ''); 
        END_IF
        IF _NominalY <= 0 THEN 
            ADSLOGSTR(ADSLOG_MSGTYPE_ERROR, 'Powod: _NominalY <= 0 (Dlugosc Nominalna to zero!)', ''); 
        END_IF
        
        bLogFired := TRUE; // Zablokuj kolejne wysyłanie
    END_IF
ELSE
    // Jeśli znowu jest poprawnie (np. poprawiono na HMI), odblokuj logi na przyszłość
    bLogFired := FALSE;
END_IF

// =========================================================
// 6. AUTO-KOREKTA KOPII I LIMITÓW DLA HMI
// =========================================================

// ZABEZPIECZENIE Z: Głębokość frezowania nie może przekroczyć grubości płyty!
_Limits.GrooveDepthZ.MaxVal := MachineConfig.RawBoardZ + 4.0;
// Bezlitosne obcięcie (clamping) wpisanej wartości do nowego limitu
_Config.GrooveDepthZ := LIMIT(_Limits.GrooveDepthZ.MinVal, _Config.GrooveDepthZ, _Limits.GrooveDepthZ.MaxVal);

IF _Config.IsValid THEN
    _Limits.RequestedCopiesX.MinVal := 1.0;
    _Limits.RequestedCopiesX.MaxVal := DINT_TO_REAL(_MaxCopiesX);
    _Limits.RequestedCopiesY.MinVal := 1.0;
    _Limits.RequestedCopiesY.MaxVal := DINT_TO_REAL(_MaxCopiesY);

    IF _Config.FillAll THEN
        _Config.RequestedCopiesX := _MaxCopiesX;
        _Config.RequestedCopiesY := _MaxCopiesY;
    ELSE
        _Config.RequestedCopiesX := LIMIT(1, _Config.RequestedCopiesX, _MaxCopiesX);
        _Config.RequestedCopiesY := LIMIT(1, _Config.RequestedCopiesY, _MaxCopiesY);
    END_IF
ELSE
    // Blokada całkowita jeśli detal się nie mieści
    _Limits.RequestedCopiesX.MinVal := 0.0;
    _Limits.RequestedCopiesX.MaxVal := 0.0;
    _Limits.RequestedCopiesY.MinVal := 0.0;
    _Limits.RequestedCopiesY.MaxVal := 0.0;
    
    _Config.RequestedCopiesX := 0;
    _Config.RequestedCopiesY := 0;
END_IF
END_METHOD

METHOD PROTECTED WriteGCodeFile : BOOL
VAR_INPUT
    sFilePath : STRING(255);
END_VAR
VAR_INST
	_iCurrentLine : INT := 1;
END_VAR
WriteGCodeFile := FALSE;

CASE _nFileWriteStep OF
    0: // INIT
        _iCurrentLine := 1; 
        _sGCodeFilePath := sFilePath;
        
        // LOG: Start operacji - wstawiamy zmienną string w miejsce %s
        ADSLOGSTR(ADSLOG_MSGTYPE_HINT, 'WriteGCode: Rozpoczynam zapis do pliku %s', _sGCodeFilePath);
        
        _nFileWriteStep := 10;

    10: // --- OTWIERANIE/TWORZENIE PLIKU ---
        fbCreateFile(
            bExecute := TRUE, 
            sPathName := _sGCodeFilePath, 
            tTimeOut := T#2S
        );
        
        IF fbCreateFile.bErr THEN 
            // LOG: Błąd tworzenia
            ADSLOGSTR(ADSLOG_MSGTYPE_ERROR, 'WriteGCode: BLAD tworzenia pliku %s!', _sGCodeFilePath);
            _nFileWriteStep := 999;
            
        ELSIF NOT fbCreateFile.bBusy THEN
            fbCreateFile(bExecute := FALSE, sPathName := _sGCodeFilePath);
            
            // LOG: Sukces tworzenia
            ADSLOGSTR(ADSLOG_MSGTYPE_HINT, 'WriteGCode: Plik utworzony pomyslnie, przechodze do zapisu.', '');
            _nFileWriteStep := 20;
        END_IF

    20: // --- ZAPISYWANIE LINII G-CODE W PĘTLI ---
        fbAppendLine(
            bExecute := TRUE, 
            sPathName := _sGCodeFilePath, 
            sBlock := _aGCodeBuffer[_iCurrentLine], 
            tTimeOut := T#2S
        );
        
        IF fbAppendLine.bErr THEN 
            // LOG: Błąd zapisu konkretnej linii
            ADSLOGSTR(ADSLOG_MSGTYPE_ERROR, 'WriteGCode: BLAD dopisywania linii G-Code!', '');
            _nFileWriteStep := 999;
            
        ELSIF NOT fbAppendLine.bBusy THEN
            fbAppendLine(bExecute := FALSE, sPathName := _sGCodeFilePath);
            
            _iCurrentLine := _iCurrentLine + 1;
            IF _iCurrentLine > _nLinesToWrite THEN
                // LOG: Koniec pętli zapisu
                ADSLOGSTR(ADSLOG_MSGTYPE_HINT, 'WriteGCode: Zapisano wszystkie linie G-Code.', '');
                _nFileWriteStep := 30; // Zapisano wszystkie linie
            END_IF
        END_IF

    30: // --- ZAMYKANIE PLIKU ---
        fbCloseFile(
            bExecute := TRUE, 
            sPathName := _sGCodeFilePath, 
            tTimeOut := T#2S
        );
        
        IF fbCloseFile.bErr THEN 
            // LOG: Błąd zamykania
            ADSLOGSTR(ADSLOG_MSGTYPE_ERROR, 'WriteGCode: BLAD zamykania pliku!', '');
            _nFileWriteStep := 999;
            
        ELSIF NOT fbCloseFile.bBusy THEN
            fbCloseFile(bExecute := FALSE, sPathName := _sGCodeFilePath);
            
            // Zapisujemy ścieżkę do struktury Config, żeby Executor NCI wiedział co odpalić
            _Config.GCodePath := _sGCodeFilePath; 
            
            // LOG: Pełny sukces
            ADSLOGSTR(ADSLOG_MSGTYPE_HINT, 'WriteGCode: Plik zamkniety pomyslnie.', '');
            _nFileWriteStep := 1000;
        END_IF

    999: // --- BŁĄD ---
        WriteGCodeFile := FALSE;
        // W tym kroku nie dajemy loga, zeby nie zaspamować konsoli błędem co każdy cykl!
        // Logi błędu wysłaliśmy tuż przed przejściem do kroku 999.

    1000: // --- GOTOWE ---
        _nFileWriteStep := 0; // Reset na przyszłość
        WriteGCodeFile := TRUE;
        
END_CASE
END_METHOD

END_FUNCTION_BLOCK

// ---- POUs/Builder/Recipes/FB_PTPBorgoFlaps.TcPOU
FUNCTION_BLOCK FB_PTPBorgoFlaps EXTENDS FB_RecipeBase

METHOD Build : BOOL
VAR_INST
    TotalY          : REAL;
    TotalX          : REAL;
    ShorterY        : REAL;
    ShorterX        : REAL;
END_VAR
_Busy := TRUE;
_Done := FALSE;
_Error := FALSE;
Build := FALSE;

THIS^.UpdateNestingLimits();

// 2. Jeśli detal wystaje poza maszynę - przerywamy od razu!
IF NOT _Config.IsValid THEN
    _Busy := FALSE;
    _Error := TRUE; 
    Build := FALSE;
    RETURN;
END_IF

// 3. Pobieramy wyliczone gabaryty nominalne do lokalnych zmiennych roboczych
TotalX   := _NominalX;
TotalY   := _NominalY; 
ShorterY := TotalY - _Config.PanelHeight;
ShorterX := TotalX - _Config.PanelHeight;


// ------------------------------------
// 1. Segregracja frezowania (Grooving)
// ------------------------------------
_SegmentsToGroove := 4;

_SegmentsGroove[1].Start.X := TotalX;
_SegmentsGroove[1].Stop.X  := 0;
_SegmentsGroove[1].Start.Y := ShorterY;
_SegmentsGroove[1].Stop.Y  := ShorterY;

_SegmentsGroove[2].Start.X := TotalX;
_SegmentsGroove[2].Stop.X  := 0; 
_SegmentsGroove[2].Start.Y := _Config.PanelHeight;
_SegmentsGroove[2].Stop.Y  := _Config.PanelHeight;

_SegmentsGroove[3].Start.X := ShorterX;
_SegmentsGroove[3].Stop.X  := ShorterX;
_SegmentsGroove[3].Start.Y := TotalY;
_SegmentsGroove[3].Stop.Y  := 0;

_SegmentsGroove[4].Start.Y := TotalY;
_SegmentsGroove[4].Stop.Y  := 0;
_SegmentsGroove[4].Start.X := _Config.PanelHeight;
_SegmentsGroove[4].Stop.X  := _Config.PanelHeight;

// ------------------------------------
// 2. Cięcie w osi X (Cut X)
// ------------------------------------
_SegmentsToCutX := 6;

// Short Box Segments
_SegmentsCutX[1].Start.X := TotalX + _Config.CuttingOverpass;
_SegmentsCutX[1].Stop.X  := ShorterX;
_SegmentsCutX[1].Start.Y := ShorterY;
_SegmentsCutX[1].Stop.Y  := ShorterY;

_SegmentsCutX[2].Start.X := _Config.PanelHeight;
_SegmentsCutX[2].Stop.X  := -_Config.CuttingOverpass;
_SegmentsCutX[2].Start.Y := ShorterY;
_SegmentsCutX[2].Stop.Y  := ShorterY;

_SegmentsCutX[3].Start.X := TotalX + _Config.CuttingOverpass;
_SegmentsCutX[3].Stop.X  := ShorterX;
_SegmentsCutX[3].Start.Y := _Config.PanelHeight;
_SegmentsCutX[3].Stop.Y  := _Config.PanelHeight;

_SegmentsCutX[4].Start.X := _Config.PanelHeight;
_SegmentsCutX[4].Stop.X  := -_Config.CuttingOverpass;
_SegmentsCutX[4].Start.Y := _Config.PanelHeight;
_SegmentsCutX[4].Stop.Y  := _Config.PanelHeight;

// Panel Dimensions 
_SegmentsCutX[5].Start.X := TotalX + _Config.CuttingOverpass;
_SegmentsCutX[5].Stop.X  := -_Config.CuttingOverpass;
_SegmentsCutX[5].Start.Y := TotalY;
_SegmentsCutX[5].Stop.Y  := TotalY;

_SegmentsCutX[6].Start.X := TotalX + _Config.CuttingOverpass;
_SegmentsCutX[6].Stop.X  := -_Config.CuttingOverpass;
_SegmentsCutX[6].Start.Y := 0;
_SegmentsCutX[6].Stop.Y  := 0;

// ------------------------------------
// 3. Cięcie w osi Y (Cut Y)
// ------------------------------------
_SegmentsToCutY := 6;

// Short Box Segments
_SegmentsCutY[1].Start.X := ShorterX;
_SegmentsCutY[1].Stop.X  := ShorterX;
_SegmentsCutY[1].Start.Y := TotalY + _Config.CuttingOverpass;
_SegmentsCutY[1].Stop.Y  := ShorterY;

_SegmentsCutY[2].Start.X := _Config.PanelHeight;
_SegmentsCutY[2].Stop.X  := _Config.PanelHeight;
_SegmentsCutY[2].Start.Y := TotalY + _Config.CuttingOverpass;
_SegmentsCutY[2].Stop.Y  := ShorterY;

_SegmentsCutY[3].Start.X := ShorterX;
_SegmentsCutY[3].Stop.X  := ShorterX;
_SegmentsCutY[3].Start.Y := _Config.PanelHeight;
_SegmentsCutY[3].Stop.Y  := -_Config.CuttingOverpass;

_SegmentsCutY[4].Start.X := _Config.PanelHeight;
_SegmentsCutY[4].Stop.X  := _Config.PanelHeight;
_SegmentsCutY[4].Start.Y := _Config.PanelHeight;
_SegmentsCutY[4].Stop.Y  := -_Config.CuttingOverpass;

// Panel Dimensions Shorter Wings
_SegmentsCutY[5].Start.X := TotalX - _Config.RailHeightCorrection;
_SegmentsCutY[5].Stop.X  := TotalX - _Config.RailHeightCorrection;
_SegmentsCutY[5].Start.Y := TotalY + _Config.CuttingOverpass;
_SegmentsCutY[5].Stop.Y  := -_Config.CuttingOverpass;

_SegmentsCutY[6].Start.X := _Config.RailHeightCorrection;
_SegmentsCutY[6].Stop.X  := _Config.RailHeightCorrection;
_SegmentsCutY[6].Start.Y := TotalY + _Config.CuttingOverpass;
_SegmentsCutY[6].Stop.Y  := -_Config.CuttingOverpass;


_Busy := FALSE;
_Done := TRUE;
Build := TRUE;
END_METHOD

METHOD PROTECTED CalculateFootprint
VAR_INPUT
END_VAR
// BorgoWings wie, że jego wymiar powiększa się o ścianki zagięcia:
_NominalX := _Config.PanelFrontWidth  + 2.0 * _Config.PanelHeight; 
_NominalY := _Config.PanelFrontLength + 2.0 * _Config.PanelHeight;
END_METHOD

PROPERTY ExecutionRoute : E_ExecutionRoute
GET
ExecutionRoute := E_ExecutionRoute.ePTP;
END_GET
END_PROPERTY

METHOD FB_init : BOOL
VAR_INPUT
	bInitRetains : BOOL; // if TRUE, the retain variables are initialized (warm start / cold start)
	bInCopyCode : BOOL;  // if TRUE, the instance afterwards gets moved into the copy code (online change)
END_VAR
_Limits.PanelFrontLength.MinVal := 100.0;
_Limits.PanelFrontLength.MaxVal := 2400.0;

_Limits.PanelFrontWidth.MinVal  := 100.0;
_Limits.PanelFrontWidth.MaxVal  := 1200.0;

_Limits.PanelHeight.MinVal      := 40.0;
_Limits.PanelHeight.MaxVal      := 100.0;

_Limits.RailHeightCorrection.MinVal := 12.0;
_Limits.RailHeightCorrection.MaxVal := 14.0;

_Limits.CuttingOverpass.MinVal := 0.0;
_Limits.CuttingOverpass.MaxVal := 50.0;

_Limits.GroovingOverpass.MinVal := 0.0;
_Limits.GroovingOverpass.MaxVal := 50.0;

_Limits.GrooveDepthZ.MinVal := 0.0;
_Limits.GrooveDepthZ.MaxVal := 9.0; //
END_METHOD

END_FUNCTION_BLOCK

// ---- POUs/Builder/Recipes/FB_PTPArona.TcPOU
FUNCTION_BLOCK FB_PTPArona EXTENDS FB_RecipeBase

METHOD Build : BOOL
VAR_INST
    TotalY          : REAL;
    TotalX          : REAL;
    ShorterY        : REAL;
    ShorterX        : REAL;
END_VAR
_Busy := TRUE;
_Done := FALSE;
_Error := FALSE;
Build := FALSE;
// 1. Zlecenie przeliczenia gabarytów, footrpintu i limitów klasie bazowej
THIS^.UpdateNestingLimits();

// 2. Jeśli detal wystaje poza maszynę - przerywamy od razu!
IF NOT _Config.IsValid THEN
    _Busy := FALSE;
    _Error := TRUE; 
    Build := FALSE;
    RETURN;
END_IF

// 3. Pobieramy wyliczone gabaryty nominalne do lokalnych zmiennych roboczych
TotalX   := _NominalX;
TotalY   := _NominalY; 

// ------------------------------------
// 1. Segregracja frezowania (Grooving)
// ------------------------------------
_SegmentsToGroove := 2;

_SegmentsGroove[1].Start.X := _Config.PanelHeight;
_SegmentsGroove[1].Stop.X  := _Config.PanelHeight;
_SegmentsGroove[1].Start.Y := TotalY;
_SegmentsGroove[1].Stop.Y  := 0;

_SegmentsGroove[2].Start.X :=  _Config.PanelHeight + 40;    
_SegmentsGroove[2].Stop.X  :=  _Config.PanelHeight + 40;    
_SegmentsGroove[2].Start.Y :=  TotalY;
_SegmentsGroove[2].Stop.Y  :=  0;                      


// ------------------------------------
// 2. Cięcie w osi X (Cut X)
// ------------------------------------+ 
_SegmentsToCutX := 2;

// Short Box Segments
_SegmentsCutX[1].Start.X := TotalX + _Config.CuttingOverpass;
_SegmentsCutX[1].Stop.X  := -_Config.CuttingOverpass;
_SegmentsCutX[1].Start.Y := 0;
_SegmentsCutX[1].Stop.Y  := 0;        

_SegmentsCutX[2].Start.X := TotalX + _Config.CuttingOverpass;                         
_SegmentsCutX[2].Stop.X  := - _Config.CuttingOverpass;                          
_SegmentsCutX[2].Start.Y := TotalY;
_SegmentsCutX[2].Stop.Y  := TotalY;        

// ------------------------------------
// 3. Cięcie w osi Y (Cut Y)
// ------------------------------------
_SegmentsToCutY := 2;

// Short Box Segments
_SegmentsCutY[1].Start.X := 0;                               
_SegmentsCutY[1].Stop.X  := 0;                               
_SegmentsCutY[1].Start.Y := TotalY +_Config.CuttingOverpass; 
_SegmentsCutY[1].Stop.Y  := -_Config.CuttingOverpass;        

_SegmentsCutY[2].Start.X := TotalX;                          
_SegmentsCutY[2].Stop.X  := TotalX;                          
_SegmentsCutY[2].Start.Y := TotalY +_Config.CuttingOverpass; 
_SegmentsCutY[2].Stop.Y  := -_Config.CuttingOverpass;        

_Busy := FALSE;
_Done := TRUE;
Build := TRUE;
END_METHOD

METHOD PROTECTED CalculateFootprint
VAR_INPUT
END_VAR
// BorgoWings wie, że jego wymiar powiększa się o ścianki zagięcia:
_NominalX := (2.0 * _Config.PanelHeight) + 40.0; 
_NominalY := _Config.PanelFrontLength;
END_METHOD

PROPERTY ExecutionRoute : E_ExecutionRoute
GET
ExecutionRoute := E_ExecutionRoute.ePTP;
END_GET
END_PROPERTY

METHOD FB_init : BOOL
VAR_INPUT
	bInitRetains : BOOL; // if TRUE, the retain variables are initialized (warm start / cold start)
	bInCopyCode : BOOL;  // if TRUE, the instance afterwards gets moved into the copy code (online change)
END_VAR
_Limits.PanelFrontLength.MinVal := 12.0;
_Limits.PanelFrontLength.MaxVal := 1234.0;

_Limits.PanelFrontWidth.MinVal  := 12.0;
_Limits.PanelFrontWidth.MaxVal  := 1234.0;

_Limits.PanelHeight.MinVal      := 12.0;
_Limits.PanelHeight.MaxVal      := 1234.0;

_Limits.RailHeightCorrection.MinVal := 12.0;
_Limits.RailHeightCorrection.MaxVal := 1234.0;

_Limits.CuttingOverpass.MinVal := 0.0;
_Limits.CuttingOverpass.MaxVal := 50.0;

_Limits.GroovingOverpass.MinVal := 0.0;
_Limits.GroovingOverpass.MaxVal := 50.0;

_Limits.GrooveDepthZ.MinVal := 0.0;
_Limits.GrooveDepthZ.MaxVal := 9.0; //
END_METHOD

END_FUNCTION_BLOCK

// ---- POUs/Builder/Recipes/FB_PTPRectangle.TcPOU
FUNCTION_BLOCK FB_PTPRectangle EXTENDS FB_RecipeBase

METHOD Build : BOOL
VAR_INST
    TotalY          : REAL;
    TotalX          : REAL;
    ShorterY        : REAL;
    ShorterX        : REAL;
END_VAR
_Busy := TRUE;
_Done := FALSE;
_Error := FALSE;
Build := FALSE;
THIS^.UpdateNestingLimits();

// 2. Jeśli detal wystaje poza maszynę - przerywamy od razu!
IF NOT _Config.IsValid THEN
    _Busy := FALSE;
    _Error := TRUE; 
    Build := FALSE;
    RETURN;
END_IF
// 3. Pobieramy wyliczone gabaryty nominalne do lokalnych zmiennych roboczych
TotalX   := _NominalX;
TotalY   := _NominalY; 

// ------------------------------------
// 1. Segregracja frezowania (Grooving)
// ------------------------------------
_SegmentsToGroove := 0;
     
// ------------------------------------
// 2. Cięcie w osi X (Cut X)
// ------------------------------------+ 
_SegmentsToCutX := 2;

// Short Box Segments
_SegmentsCutX[1].Start.X := TotalX + _Config.CuttingOverpass;
_SegmentsCutX[1].Stop.X  := -_Config.CuttingOverpass;
_SegmentsCutX[1].Start.Y := 0;
_SegmentsCutX[1].Stop.Y  := 0;        

_SegmentsCutX[2].Start.X := TotalX + _Config.CuttingOverpass;                         
_SegmentsCutX[2].Stop.X  := - _Config.CuttingOverpass;                          
_SegmentsCutX[2].Start.Y := TotalY;
_SegmentsCutX[2].Stop.Y  := TotalY;        

// ------------------------------------
// 3. Cięcie w osi Y (Cut Y)
// ------------------------------------
_SegmentsToCutY := 2;

// Short Box Segments
_SegmentsCutY[1].Start.X := 0;                               
_SegmentsCutY[1].Stop.X  := 0;                               
_SegmentsCutY[1].Start.Y := TotalY +_Config.CuttingOverpass; 
_SegmentsCutY[1].Stop.Y  := -_Config.CuttingOverpass;        

_SegmentsCutY[2].Start.X := TotalX;                          
_SegmentsCutY[2].Stop.X  := TotalX;                          
_SegmentsCutY[2].Start.Y := TotalY +_Config.CuttingOverpass; 
_SegmentsCutY[2].Stop.Y  := -_Config.CuttingOverpass;        

_Busy := FALSE;
_Done := TRUE;
Build := TRUE;
END_METHOD

METHOD PROTECTED CalculateFootprint
VAR_INPUT
END_VAR
_NominalX := _Config.PanelFrontWidth;
_NominalY := _Config.PanelFrontLength;
END_METHOD

PROPERTY ExecutionRoute : E_ExecutionRoute
GET
ExecutionRoute := E_ExecutionRoute.ePTP;
END_GET
END_PROPERTY

METHOD FB_init : BOOL
VAR_INPUT
	bInitRetains : BOOL; // if TRUE, the retain variables are initialized (warm start / cold start)
	bInCopyCode : BOOL;  // if TRUE, the instance afterwards gets moved into the copy code (online change)
END_VAR
_Limits.PanelFrontLength.MinVal := 12.0;
_Limits.PanelFrontLength.MaxVal := 2400.0;

_Limits.PanelFrontWidth.MinVal  := 12.0;
_Limits.PanelFrontWidth.MaxVal  := 1200.0;

_Limits.PanelHeight.MinVal      := 12.0;
_Limits.PanelHeight.MaxVal      := 1234.0;

_Limits.RailHeightCorrection.MinVal := 12.0;
_Limits.RailHeightCorrection.MaxVal := 13.0;

_Limits.CuttingOverpass.MinVal := 0.0;
_Limits.CuttingOverpass.MaxVal := 50.0;

_Limits.GroovingOverpass.MinVal := 0.0;
_Limits.GroovingOverpass.MaxVal := 50.0;

_Limits.GrooveDepthZ.MinVal := 0.0;
_Limits.GrooveDepthZ.MaxVal := 9.0; //
END_METHOD

END_FUNCTION_BLOCK

// ---- POUs/Builder/Recipes/FB_NCICircle.TcPOU
FUNCTION_BLOCK FB_NCICircle EXTENDS FB_RecipeBase

METHOD Build : BOOL
VAR
      i          : INT;
END_VAR

VAR_INST
    nBuildStep : INT;
    machineConfig : ST_GantryXYZ_Config;
END_VAR
Build := FALSE;

CASE nBuildStep OF
    0:
        _Busy := TRUE;
        _Done := FALSE;
        _Error := FALSE;
        _nLinesToWrite := 0;
        
        ADSLOGSTR(ADSLOG_MSGTYPE_HINT, 'Generator: Budowanie G-Code (Z=8, F1500)', '');
        
        THIS^.UpdateNestingLimits();
        IF NOT _Config.IsValid THEN
            ADSLOGSTR(ADSLOG_MSGTYPE_ERROR, 'NCIBuilder: Walidacja nie przeszla! Ustawiam ERROR.', '');
            _Busy := FALSE;
            _Error := TRUE;
            Build := FALSE;
            RETURN;
        END_IF
        
        // --- BUFOR G-CODE ---
        _aGCodeBuffer[1]   := '(1001)$N';
        _aGCodeBuffer[2]   := 'N0 G01 X16.005 Y43.953 Z28 F400$N';
        _aGCodeBuffer[3]   := 'N1 G01 Q1=-180. F12000$N';
        _aGCodeBuffer[4]   := 'N2 G01 Z8 F400$N';
        _aGCodeBuffer[5]   := 'N3 Y12.093 F1500$N';
        _aGCodeBuffer[6]   := 'N4 G01 Z18 F400$N';
        _aGCodeBuffer[7]   := 'N5 G01 Q1=-90. F12000$N';
        _aGCodeBuffer[8]   := 'N6 G01 Z8 F400$N';
        _aGCodeBuffer[9]   := 'N7 X19.995 F1500$N';
        _aGCodeBuffer[10]  := 'N8 G01 Z18 F400$N';
        _aGCodeBuffer[11]  := 'N9 G01 Q1=0. F12000$N';
        _aGCodeBuffer[12]  := 'N10 G01 Z8 F400$N';
        _aGCodeBuffer[13]  := 'N11 Y92.083 F1500$N';
        _aGCodeBuffer[14]  := 'N12 G01 Z18 F400$N';
        _aGCodeBuffer[15]  := 'N13 G01 Q1=90. F12000$N';
        _aGCodeBuffer[16]  := 'N14 G01 Z8 F400$N';
        _aGCodeBuffer[17]  := 'N15 X16.005 F1500$N';
        _aGCodeBuffer[18]  := 'N16 G01 Z18 F400$N';
        _aGCodeBuffer[19]  := 'N17 G01 Q1=180. F12000$N';
        _aGCodeBuffer[20]  := 'N18 G01 Z8 F400$N';
        _aGCodeBuffer[21]  := 'N19 Y43.953 F1500$N';
        _aGCodeBuffer[22]  := 'N20 Z18 F400$N';
        _aGCodeBuffer[23]  := 'N21 X54.021 Y72.79 F2000$N';
        _aGCodeBuffer[24]  := 'N22 G01 Q1=90. F12000$N';
        _aGCodeBuffer[25]  := 'N23 G01 Z8 F400$N';
        _aGCodeBuffer[26]  := 'N24 G03 Y36.8 Q1=270. J-17.995 F1500$N';
        _aGCodeBuffer[27]  := 'N25 Y72.79 Q1=450. J17.995 F1500$N';
        _aGCodeBuffer[28]  := 'N26 G01 Z18 F400$N';
        _aGCodeBuffer[29]  := 'N27 X96.443 Y63.279 F2000$N';
        _aGCodeBuffer[30]  := 'N28 G01 Q1=360. F12000$N';
        _aGCodeBuffer[31]  := 'N29 G01 Z8 F400$N';
        _aGCodeBuffer[32]  := 'N30 Y79.328 F1500$N';
        _aGCodeBuffer[33]  := 'N31 G01 Z18 F400$N';
        _aGCodeBuffer[34]  := 'N32 G01 Q1=270.026 F12000$N';
        _aGCodeBuffer[35]  := 'N33 G01 Z8 F400$N';
        _aGCodeBuffer[36]  := 'N34 X107.344 Y79.333 F1500$N';
        _aGCodeBuffer[37]  := 'N35 G01 Z18 F400$N';
        _aGCodeBuffer[38]  := 'N36 G01 Q1=191.577 F12000$N';
        _aGCodeBuffer[39]  := 'N37 G01 Z8 F400$N';
        _aGCodeBuffer[40]  := 'N38 X108.339 Y74.477 F1500$N';
        _aGCodeBuffer[41]  := 'N39 Q1=195.179 F12000$N';
        _aGCodeBuffer[42]  := 'N40 X109.637 Y69.693 F1500$N';
        _aGCodeBuffer[43]  := 'N41 Q1=198.781 F12000$N';
        _aGCodeBuffer[44]  := 'N42 X111.233 Y64.999 F1500$N';
        _aGCodeBuffer[45]  := 'N43 Q1=202.383 F12000$N';
        _aGCodeBuffer[46]  := 'N44 X113.12 Y60.416 F1500$N';
        _aGCodeBuffer[47]  := 'N45 Q1=205.985 F12000$N';
        _aGCodeBuffer[48]  := 'N46 X115.292 Y55.96 F1500$N';
        _aGCodeBuffer[49]  := 'N47 Q1=209.587 F12000$N';
        _aGCodeBuffer[50]  := 'N48 X117.74 Y51.649 F1500$N';
        _aGCodeBuffer[51]  := 'N49 Q1=213.188 F12000$N';
        _aGCodeBuffer[52]  := 'N50 X120.453 Y47.501 F1500$N';
        _aGCodeBuffer[53]  := 'N51 Q1=216.79 F12000$N';
        _aGCodeBuffer[54]  := 'N52 X123.422 Y43.531 F1500$N';
        _aGCodeBuffer[55]  := 'N53 Q1=222.811 F12000$N';
        _aGCodeBuffer[56]  := 'N54 G02 X124.082 Y41.639 Q1=175.653 I-1.838 J-1.703 F1500$N';
        _aGCodeBuffer[57]  := 'N55 G01 Q1=179.901 F12000$N';
        _aGCodeBuffer[58]  := 'N56 G02 X122.726 Y33.034 Q1=162.194 I-28.298 J0.049 F1500$N';
        _aGCodeBuffer[59]  := 'N57 G01 Q1=153.406 F12000$N';
        _aGCodeBuffer[60]  := 'N58 G02 X104.492 Y27.546 Q1=60.095 I-11.707 J5.861 F1500$N';
        _aGCodeBuffer[61]  := 'N59 G01 Q1=64.069 F12000$N';
        _aGCodeBuffer[62]  := 'N60 G02 X98.805 Y33.393 Q1=24.352 I5.25 J10.797 F1500$N';
        _aGCodeBuffer[63]  := 'N61 G01 Q1=17.533 F12000$N';
        _aGCodeBuffer[64]  := 'N62 G02 X97.527 Y43.068 Q1=-2.484 I26.774 J8.458 F1500$N';
        _aGCodeBuffer[65]  := 'N63 G01 Q1=3.871 F12000$N';
        _aGCodeBuffer[66]  := 'N64 G02 X96.468 Y63.28 Q1=2.127 I663.315 J44.884 F1500$N';
        _aGCodeBuffer[67]  := 'N65 G01 Z18 F400$N';
        _aGCodeBuffer[68]  := 'N66 G01 Q1=92.125 F12000$N';
        _aGCodeBuffer[69]  := 'N67 G01 Z8 F400$N';
        _aGCodeBuffer[70]  := 'N68 X96.443 Y63.279 Z16.002 F400$N';
        _aGCodeBuffer[71]  := 'N69 Z18 F400$N';
        _aGCodeBuffer[72]  := 'N70 X151.232 Y45.688 F2000$N';
        _aGCodeBuffer[73]  := 'N71 G01 Q1=180. F12000$N';
        _aGCodeBuffer[74]  := 'N72 G01 Z8 F400$N';
        _aGCodeBuffer[75]  := 'N73 Y34.904 F1500$N';
        _aGCodeBuffer[76]  := 'N74 G01 Z18 F400$N';
        _aGCodeBuffer[77]  := 'N75 G01 Q1=270. F12000$N';
        _aGCodeBuffer[78]  := 'N76 G01 Z8 F400$N';
        _aGCodeBuffer[79]  := 'N77 X271.222 F1500$N';
        _aGCodeBuffer[80]  := 'N78 G01 Z18 F400$N';
        _aGCodeBuffer[81]  := 'N79 G01 Q1=360. F12000$N';
        _aGCodeBuffer[82]  := 'N80 G01 Z8 F400$N';
        _aGCodeBuffer[83]  := 'N81 Y54.894 F1500$N';
        _aGCodeBuffer[84]  := 'N82 G01 Z18 F400$N';
        _aGCodeBuffer[85]  := 'N83 G01 Q1=450. F12000$N';
        _aGCodeBuffer[86]  := 'N84 G01 Z8 F400$N';
        _aGCodeBuffer[87]  := 'N85 X151.232 F1500$N';
        _aGCodeBuffer[88]  := 'N86 G01 Z18 F400$N';
        _aGCodeBuffer[89]  := 'N87 G01 Q1=540. F12000$N';
        _aGCodeBuffer[90]  := 'N88 G01 Z8 F400$N';
        _aGCodeBuffer[91]  := 'N89 Y45.688 F1500$N';
        _aGCodeBuffer[92]  := 'N90 Z18 F400$N';
        _aGCodeBuffer[93]  := 'N91 X85.221 Y188.878 F2000$N';
        _aGCodeBuffer[94]  := 'N92 G01 Q1=450. F12000$N';
        _aGCodeBuffer[95]  := 'N93 G01 Z8 F400$N';
        _aGCodeBuffer[96]  := 'N94 G03 Y98.888 Q1=630. J-44.995 F1500$N';
        _aGCodeBuffer[97]  := 'N95 Y188.878 Q1=810. J44.995 F1500$N';
        _aGCodeBuffer[98]  := 'N96 G01 Z18 F400$N';
        _aGCodeBuffer[99]  := 'N97 X173.205 Y149.704 F2000$N';
        _aGCodeBuffer[100] := 'N98 G01 Q1=900. F12000$N';
        _aGCodeBuffer[101] := 'N99 G01 Z8 F400$N';
        _aGCodeBuffer[102] := 'N100 Y108.883 F1500$N';
        _aGCodeBuffer[103] := 'N101 G03 X183.2 Y98.888 Q1=990. I9.995 F1500$N';
        _aGCodeBuffer[104] := 'N102 G01 X253.2 F1500$N';
        _aGCodeBuffer[105] := 'N103 G03 X263.195 Y108.883 Q1=1080. J9.995 F1500$N';
        _aGCodeBuffer[106] := 'N104 G01 Y178.883 F1500$N';
        _aGCodeBuffer[107] := 'N105 G03 X253.2 Y188.878 Q1=1170. I-9.995 F1500$N';
        _aGCodeBuffer[108] := 'N106 G01 X183.2 F1500$N';
        _aGCodeBuffer[109] := 'N107 G03 X173.205 Y178.883 Q1=1260. J-9.995 F1500$N';
        _aGCodeBuffer[110] := 'N108 G01 Y149.704 F1500$N';
        _aGCodeBuffer[111] := 'N109 Z18 F400$N';
        _aGCodeBuffer[112] := 'N110 X296.995 Y178.706 F2000$N';
        _aGCodeBuffer[113] := 'N111 G01 Q1=1080. F12000$N';
        _aGCodeBuffer[114] := 'N112 G01 Z8 F400$N';
        _aGCodeBuffer[115] := 'N113 Y190 F1500$N';
        _aGCodeBuffer[116] := 'N114 G03 X277 Y209.995 Q1=1170. I-19.995 F1500$N';
        _aGCodeBuffer[117] := 'N115 G01 X20 F1500$N';
        _aGCodeBuffer[118] := 'N116 G03 X0.005 Y190 Q1=1260. J-19.995 F1500$N';
        _aGCodeBuffer[119] := 'N117 G01 Y20 F1500$N';
        _aGCodeBuffer[120] := 'N118 G03 X20 Y0.005 Q1=1350. I19.995 F1500$N';
        _aGCodeBuffer[121] := 'N119 G01 X277 F1500$N';
        _aGCodeBuffer[122] := 'N120 G03 X296.995 Y20 Q1=1440. J19.995 F1500$N';
        _aGCodeBuffer[123] := 'N121 G01 Y178.706 F1500$N';
        _aGCodeBuffer[124] := 'N122 Z18 F400$N';
        _aGCodeBuffer[125] := 'N123 Z28 F400$N';
        _aGCodeBuffer[126] := 'N124 G01 Z18 F400$N';
        
        _nLinesToWrite := 126; 
        
        // Czyszczenie reszty bufora
        FOR i := (_nLinesToWrite + 1) TO 200 DO 
            _aGCodeBuffer[i] := '';
        END_FOR
        
        nBuildStep := 10;

